// TwinCAT 3 PLC project DMAX
// Title: CalmarProdDmax
// Company: WIFAG-Polytype
// Author: Wifag//Polytype
// ProjectVersion: 2.0.2.24
// Description: All rights reserved (c) Wifag//Polytype, Fribourg/Switzerland (2021)
// ProgramVersion: 3.1.4023.0
// CompilerDefines: checks_in_libs
// libraries:
//   CalmarCommons, * (WIFAG-Polytype)
//   CalmarCompDevices, * (WIFAG-Polytype)
//   CalmarCompPrint, * (WIFAG-Polytype)
//   CalmarCompSystem, * (WIFAG-Polytype)
//   CalmarCompTcpIp, * (WIFAG-Polytype)
//   Tc2_EtherCAT, * (Beckhoff Automation GmbH)
//   Tc2_Math, * (Beckhoff Automation GmbH)
//   Tc2_Standard, * (Beckhoff Automation GmbH)
//   Tc2_System, * (Beckhoff Automation GmbH)
//   Tc2_TcpIp, * (Beckhoff Automation GmbH)
//   Tc2_Utilities, * (Beckhoff Automation GmbH)
//   Tc3_JsonXml, * (Beckhoff Automation GmbH)
//   VisuDialogs, * (System)
// project tree:
//   DUTs/Camera/ EN_CAMERA_TEACH.TcDUT, E_CameraDevice.TcDUT, E_CameraMode.TcDUT, E_DeformationType.TcDUT, ST_ADS_CAMERA.TcDUT, ST_CameraPoint.TcDUT, ST_CAMERA_CORRECTION_QV.TcDUT, ST_CAMERA_RESULT.TcDUT, ST_CAMERA_TEACH_QV.TcDUT, ST_CORRECTION_POINT.TcDUT, ST_TeachPoint.TcDUT
//   DUTs/ EN_MSG_LIST.TcDUT
//   / GlobalTextList.TcGTLO, Visualization Manager.TcVMO (not stored)
//   GVLs/ EC_DefGrid.TcGVL, GVL_Camera.TcGVL, GVL_Deformation.TcGVL
//   POUs/Machine/ExhaustSystem/ FB_ExhaustSystemPrint.TcPOU, _VISU_ExhaustSystemPrint.TcVIS
//   POUs/Machine/PowerControl/ FB_PowerControl.TcPOU, _VISU_PowerControl.TcVIS
//   POUs/Machine/UV_LED_Modul/ FB_UvLedModule.TcPOU, _VISU_UvLedModule.TcVIS
//   POUs/Print/Ads/ FB_ADS_CAMERA.TcPOU, FB_ADS_DVTSHEETALIGNMENT.TcPOU
//   POUs/Print/Camera/ FB_CameraBase.TcPOU, FB_CameraDummy.TcPOU, FB_CameraTcpIp.TcPOU, FB_CameraTrigger.TcPOU, FB_LineCamera.TcPOU, FB_LineCamera106.TcPOU, FB_LineCamera76.TcPOU, FB_MarkCamera.TcPOU, FB_SystronCamera.TcPOU, FB_TcpIpComm.TcPOU, F_DeformationPointAcc_ToString.TcPOU, F_CamPoint_ToString.TcPOU, ImagePool.TcIPO (not stored), I_Camera.TcIO, I_CameraSink.TcIO, I_CameraTrigger.TcIO, I_CameraTriggerDevice.TcIO, _VISU_CameraBase.TcVIS, _VISU_CameraBaseSetting.TcVIS, _VISU_CameraTcpIp.TcVIS, _VISU_CameraTcpIpSetting.TcVIS, _VISU_CameraTrigger.TcVIS, _VISU_DeformationPoint.TcVIS, _VISU_LineCamera.TcVIS, _VISU_MarkCamera.TcVIS (not stored), _VISU_SystronCamera.TcVIS
//   POUs/Print/DefGrid/ E_DeformationStep.TcTLEO, FB_ContainerDefGrid.TcPOU, FB_CTManagerDefGrid.TcPOU, FB_DeformationPointFIFO.TcPOU, FB_DropSpeedComp.TcPOU, FB_FineAlignement.TcPOU, FB_ImageDeformation.TcPOU, FB_DefGridParamMediator.TcPOU, FB_PointCorr.TcPOU, FB_PrintOverview.TcPOU, FB_PrintPositionDmax.TcPOU, FB_ProdManager_DMAX.TcPOU, FB_PythonDeformation.TcPOU, FB_PythonInterface.TcPOU, FB_StartPositionDummy.TcPOU, FB_WorkerDefGrid.TcPOU, FB_WorkerDefGrid_Camera.TcPOU, FB_WorkerDefGrid_Deformation.TcPOU, FB_WorkerDefGrid_Delete.TcPOU, FB_WorkerDefGrid_Print.TcPOU, FB_WorkerDefGrid_Python.TcPOU, FB_WorkerDefGrid_Verify.TcPOU, F_EncoderSpeedComp.TcPOU, F_MeterToSubPixelReal.TcPOU (not stored), I_DeformationHandler.TcIO, I_GridPointCorrection.TcIO, I_ParamMediator.TcIO, I_ProdManager.TcIO, ST_CameraGridSettings.TcDUT, ST_CameraPointTbl.TcDUT (not stored), ST_DeformationPointTbl.TcDUT, ST_WorkerDefGrid_CTData.TcDUT
//   POUs/Print/DefGrid/_Test/ E_GridTypeSelection.TcTLEO, Txt_GridTypeSelection.TcTLO
//   POUs/Print/DefGrid/_VISU_Templates/ E_DeformationType.TcTLO, _VISU_ContainerDefGrid.TcVIS, _VISU_CTsFlow.TcVIS, _VISU_DefGridTable.TcVIS, _VISU_FineAlignment.TcVIS, _VISU_GridPointView.TcVIS (not stored), _VISU_ImageDeformation.TcVIS (not stored), _VISU_PlacementXY.TcVIS (not stored), _VISU_PlacementXY_cross.TcVIS (not stored), _VISU_PrintPositionDmax.TcVIS (not stored), _VISU_DropSpeedComp_Setup.TcVIS, _VISU_StartPositionDummy.TcVIS (not stored), _VISU_WorkerDefGrid.TcVIS (not stored), _VISU_WorkerDefGrid_Camera.TcVIS (not stored), _VISU_WorkerDefGrid_Deformation.TcVIS (not stored), _VISU_WorkerDefGrid_Delete.TcVIS (not stored), _VISU_WorkerDefGrid_Print.TcVIS (not stored), _VISU_WorkerDefGrid_Python.TcVIS (not stored), _VISU_WorkerDefGrid_small.TcVIS (not stored), _VISU_WorkerDefGrid_Verify.TcVIS (not stored)
//   POUs/Print/ FB_SheetDetectSupervision.TcPOU, ST_SheetDetectSupervisionPar.TcDUT
//   Version/ Global_Version.TcGVL

// ---- DUTs/Camera/EN_CAMERA_TEACH.TcDUT
TYPE EN_CAMERA_TEACH :
(*************************************************************************************************)
(*  FILENAME:    EN_CAMERA_TEACH                                                                 *)
(*  PROJECT:     CALMAR PUPLC                                                                    *)
(*  COPYRIGHT:   All rights reserved (c) Wifag//Polytype, Fribourg/Switzerland (2018)            *)
(*  ENVIRONMENT: TwinCAT PLC                                                                     *)
(*  VERSION:     <version>                                                                       *)
(*************************************************************************************************)
(*  DESCRIPTION:                                                                   <description> *)
(*    Enumeration for camera teach.                                                              *)
(*                                                                                </description> *)
(*************************************************************************************************)

(
  eTeachInit         := 0,
  eTeachStart        := 1,
  eTeachCompleted    := 2,
  eTeachCanceled     := 3,
  eTeachError        := 4
);
END_TYPE

// ---- DUTs/Camera/E_CameraDevice.TcDUT
{attribute 'qualified_only'}
{attribute 'strict'}
{attribute 'to_string'}
TYPE E_CameraDevice :
(
  SheetDetect              := 0,   // SheetDetect
  PrintMark                := 1,   // PrintMark
  Scanner                  := 2,   // Scanner
  ScannerWithoutBackground := 3    // ScannerWithoutBackground
);
END_TYPE

// ---- DUTs/Camera/E_CameraMode.TcDUT
{attribute 'qualified_only'}
{attribute 'strict'}
{attribute 'to_string'}
TYPE E_CameraMode :
(
  NoCorrection := 0,   // NoCorrection
  XYR          := 1,   // XYR
  Live         := 2,   // Live deformation
  Trend        := 3,   // Live deformation with trend
  Auto         := 4    // Auto
);
END_TYPE

// ---- DUTs/Camera/E_DeformationType.TcDUT
{attribute 'qualified_only'}
{attribute 'to_string'}
TYPE E_DeformationType :
(
  NoDeformation   := 0,   // NoCorrection
  ScriptGrid      := 1,   // Py script (live)
  ScriptGridTrend := 2,   // Py script (live with trend)
  LocalMarks1D    := 3    // Plc generated with 1D marks
)  UINT;
END_TYPE

// ---- DUTs/Camera/ST_ADS_CAMERA.TcDUT
TYPE ST_ADS_CAMERA :
(*************************************************************************************************)
(*  FILENAME:    ST_ADS_CAMERA                                                                   *)
(*  PROJECT:     CALMAR PUPLC                                                                    *)
(*  COPYRIGHT:   All rights reserved (c) Wifag//Polytype, Fribourg/Switzerland (2018)            *)
(*  ENVIRONMENT: TwinCAT PLC                                                                     *)
(*  VERSION:     <version>                                                                       *)
(*************************************************************************************************)
(*  DESCRIPTION:                                                                   <description> *)
(*    ADS structure for camera (Systron, QualiVision).                                           *)
(*                                                                                </description> *)
(*************************************************************************************************)

STRUCT
  iO_Version                : UINT    := 010300;  (*1.3.0*)
  aO_Type                   : STRING := 'Camera';
  aO_Name                   : STRING := 'Camera';
  sO_Message                : ST_ADS_MSG_IF;

  (*In*)
  bI_Enable                 : BOOL := TRUE;      (*Enable this device*)

  eI_CameraDevice           : E_CameraDevice;    (*Camera device*)
  eI_CameraMode             : E_CameraMode;      (*Camera mode*)

  eI_TeachProgress          : EN_CAMERA_TEACH;   (*Teach progress*)
  sI_TeachPointsQV          : ARRAY[1..GVL_Camera.cC_QUALIVISION_MAX_NB_MARKS] OF ST_CAMERA_TEACH_QV;
  
  sI_CorrectionPointIndication: ARRAY[1..4] OF ST_CORRECTION_POINT;

  (*Out*)
  iO_MaxNbMarksQV           : INT := GVL_Camera.cC_QUALIVISION_MAX_NB_MARKS; 
  sO_PointsReadQV           : ST_COMMAND_PLC;    (*New points read by QualiVision*)
  iO_AvailableNbReadPointQV : INT; 
  sO_ReadPointsQV           : ARRAY[1..GVL_Camera.cC_QUALIVISION_MAX_NB_MARKS] OF ST_CAMERA_CORRECTION_QV;

END_STRUCT
END_TYPE

// ---- DUTs/Camera/ST_CameraPoint.TcDUT
TYPE ST_CameraPoint :
STRUCT
  (*Valus from camera [px/4800dpi]*)
  id                  : UDINT := 0;     (*mark id*)
  x_ref               : DINT := 0;      (*Referenz x deviation [px/4800dpi]*)
  y_ref               : DINT := 0;      (*Referenz y deviation [px/4800dpi]*)
  lx                  : DINT := 0;      (*Referenz in picture x deviation [px/4800dpi]*)
  ly                  : DINT := 0;      (*Referenz in picture y deviation [px/4800dpi]*)
  valid               : BOOL := FALSE;  (*TRUE = PASS, FALSE = FAIL*)
  x                   : DINT := 0;      (*x deviation [px/4800dpi]*)
  y                   : DINT := 0;      (*y deviation [px/4800dpi]*)
END_STRUCT
END_TYPE

// ---- DUTs/Camera/ST_CAMERA_CORRECTION_QV.TcDUT
TYPE ST_CAMERA_CORRECTION_QV :
(*************************************************************************************************)
(*  FILENAME:    ST_CAMERA_CORRECTION_QV                                                         *)
(*  PROJECT:     CALMAR PUPLC                                                                    *)
(*  COPYRIGHT:   All rights reserved (c) Wifag//Polytype, Fribourg/Switzerland (2016)            *)
(*  ENVIRONMENT: TwinCAT PLC                                                                     *)
(*  VERSION:     <version>                                                                       *)
(*************************************************************************************************)
(*  DESCRIPTION:                                                                   <description> *)
(*    Correction of smart camera QualiVision for PUC.                                            *)
(*                                                                                </description> *)
(*************************************************************************************************)

STRUCT
  (*PUC correction points [mm]*)
  valid               : BOOL := FALSE;  (*TRUE = PASS, FALSE = FAIL*)
  PaddingByte01       : BYTE;           (*PUC needs it for stream reading. TC3 uses 8 byte alignment.*)
  PaddingByte02       : BYTE;           (*PUC needs it for stream reading. TC3 uses 8 byte alignment.*)
  PaddingByte03       : BYTE;           (*PUC needs it for stream reading. TC3 uses 8 byte alignment.*)
  x_origin            : REAL := 0;      (*Referenz x origin [mm]*)
  y_origin            : REAL := 0;      (*Referenz y origin [mm]*)
  x_correction        : REAL := 0;      (*x correction [mm]*)
  y_correction        : REAL := 0;      (*y correction [mm]*)
  PaddingBytes04      : REAL;           (*PUC needs it for stream reading. TC3 uses 8 byte alignment.*)
END_STRUCT
END_TYPE

// ---- DUTs/Camera/ST_CAMERA_RESULT.TcDUT
TYPE ST_CAMERA_RESULT :
(*************************************************************************************************)
(*  FILENAME:    ST_CAMERA_RESULT.EXP                                                            *)
(*  PROJECT:     CALMAR PUPLC                                                                    *)
(*  COPYRIGHT:   All rights reserved (c) Wifag//Polytype, Fribourg/Switzerland (2016)            *)
(*  ENVIRONMENT: TwinCAT PLC                                                                     *)
(*  VERSION:     <version>                                                                       *)
(*************************************************************************************************)
(*  DESCRIPTION:                                                                   <description> *)
(*    Output of smart camera Systron.                                                            *)
(*                                                                                </description> *)
(*************************************************************************************************)

STRUCT
  x_ref               : REAL := 0;      (*Referenz x deviation [mm]*)
  y_ref               : REAL := 0;      (*Referenz y deviation [mm]*)
  valid               : BOOL := TRUE;   (*TRUE = PASS, FALSE = FAIL*)
  x                   : REAL := 0;      (*x deviation [mm]*)
  y                   : REAL := 0;      (*y deviation [mm]*)
END_STRUCT
END_TYPE

// ---- DUTs/Camera/ST_CAMERA_TEACH_QV.TcDUT
TYPE ST_CAMERA_TEACH_QV :
(*************************************************************************************************)
(*  FILENAME:    ST_CAMERA_TEACH_QV                                                              *)
(*  PROJECT:     CALMAR PUPLC                                                                    *)
(*  COPYRIGHT:   All rights reserved (c) Wifag//Polytype, Fribourg/Switzerland (2016)            *)
(*  ENVIRONMENT: TwinCAT PLC                                                                     *)
(*  VERSION:     <version>                                                                       *)
(*************************************************************************************************)
(*  DESCRIPTION:                                                                   <description> *)
(*    Teach points for smart camera QualiVision from PUC.                                        *)
(*                                                                                </description> *)
(*************************************************************************************************)

STRUCT
  x_ref_Print         : REAL := 0;      (*Referenz x deviation [mm]*)
  y_ref_Print         : REAL := 0;      (*Referenz y deviation [mm]*)
END_STRUCT
END_TYPE

// ---- DUTs/Camera/ST_CORRECTION_POINT.TcDUT
TYPE ST_CORRECTION_POINT :
(*************************************************************************************************)
(*  FILENAME:    ST_CORRECTION_POINT                                                             *)
(*  PROJECT:     CALMAR PUPLC                                                                    *)
(*  COPYRIGHT:   All rights reserved (c) Wifag//Polytype, Fribourg/Switzerland (2021)            *)
(*  ENVIRONMENT: TwinCAT PLC                                                                     *)
(*  VERSION:     <version>                                                                       *)
(*************************************************************************************************)
(*  DESCRIPTION:                                                                   <description> *)
(*    PUC correction point indication provided from job, written at print start.                 *)
(*                                                                                </description> *)
(*************************************************************************************************)

STRUCT
  x        : REAL := 0;      (*Correction indication x [mm]*)
  y        : REAL := 0;      (*Correction indication y [mm]*)
  posx     : REAL := 0;      (*Correction location in x [mm]*)
  posy     : REAL := 0;      (*Correction location in y [mm]*)
END_STRUCT
END_TYPE

// ---- DUTs/Camera/ST_TeachPoint.TcDUT
TYPE ST_TeachPoint :
STRUCT
  (*Valus for printer [mm]*)
  id                  : UDINT;           (*point id*)
  x_ref_Print         : LREAL := 0;      (*Referenz x deviation [mm]*)
  y_ref_Print         : LREAL := 0;      (*Referenz y deviation [mm]*)
  x_teach_Print       : LREAL := 0;      (*Teach x deviation [mm]*)
  y_teach_Print       : LREAL := 0;      (*Teach y deviation [mm]*)
  x_Print             : LREAL := 0;      (*x deviation [mm]*)
  y_Print             : LREAL := 0;      (*y deviation [mm]*)
  valid               : BOOL  := FALSE;  (**)
END_STRUCT
END_TYPE

// ---- DUTs/EN_MSG_LIST.TcDUT
TYPE EN_MSG_LIST :
(*************************************************************************************************)
(*  FILENAME:    EN_MSG_LIST.EXP                                                                 *)
(*  PROJECT:     CALMAR PUPLC                                                                    *)
(*  COPYRIGHT:   All rights reserved (c) Wifag//Polytype, Fribourg/Switzerland (2016)            *)
(*  ENVIRONMENT: TwinCAT PLC                                                                     *)
(*  VERSION:     <version>                                                                       *)
(*************************************************************************************************)
(*  DESCRIPTION:                                                                   <description> *)
(*     This block containts the global list for all messages used by `FB_MESSAGE`.               *)
(*                                                                                </description> *)
(*************************************************************************************************)
(
  // start at                       eCStag_MSG_BASE := 10000,
  eC_STAG_CAM_NOTAVAIL                              :=10000,  (*CameraNotAvailable*)
  eC_STAG_CAM_MODE_NOTSUPPORTED                     :=10001,  (*CameraModeNotSupported*)
  eC_STAG_CAM_NOTENGOUGH_TEACH_POINTS               :=10002,  (*CameraNotEnoughTeachPoints*)
  eC_STAG_DEF_SCRIPT_NOT_RUNNING                    :=10003,  (*DeformationScriptNotRunning*)
  eC_STAG_CAM_TEACH_ERROR                           :=10004,  (*CameraTeachError*)
  eC_STAG_IMAGELENGTH_NOT_SUPPORTED                 :=10005,  (*ImageLengthNotSupported*)
  eC_STAG_DEFORMATION_LIMITED                       :=10006   (*DeformationWasLimited (Warning)*)
);
END_TYPE

// ---- POUs/Print/DefGrid/E_DeformationStep.TcTLEO
{attribute 'qualified_only'}
{attribute 'strict'}
{attribute 'to_string'}
TYPE E_DeformationStep :
(
  nothing := 0,
  createdScriptContainer := 1,
  cameraStarted := 2,
  cameraDone := 3,
  gridStarted := 4
);
END_TYPE

// ---- POUs/Print/DefGrid/ST_CameraGridSettings.TcDUT
TYPE ST_CameraGridSettings :
STRUCT
  bValid            : BOOL;   // ?
  eCameraMode       : E_CameraMode;
  eDeformationType  : E_DeformationType;  // selected deformation type based on selecte camera and settings
  fGridFeaturePitch : LREAL;  // feature grid picth (cam frame width) [px]
  fDetectToCam      : LREAL;  // distance between detection and camera [m]
END_STRUCT
END_TYPE

// ---- POUs/Print/DefGrid/ST_DeformationPointTbl.TcDUT
(*
  Table representation of a point
*)
TYPE ST_DeformationPointTbl :
STRUCT
  bSet          : BOOL;
  tTime         : T_DCTIME64;
  sPoint        : ST_DeformationPointAccurate;
END_STRUCT
END_TYPE

// ---- POUs/Print/DefGrid/ST_WorkerDefGrid_CTData.TcDUT
// workers additional data for all attached CTs
TYPE ST_WorkerDefGrid_CTData :
STRUCT
  fPosRelToAttach : LREAL;    // ct relative position to attach
  nChargedCols : UDINT;       // number of streamed columns of this ct
  nXS : DINT;                 // XS print start position
END_STRUCT
END_TYPE

// ---- POUs/Print/DefGrid/_Test/E_GridTypeSelection.TcTLEO
{attribute 'qualified_only'}
{attribute 'strict'}
{attribute 'to_string'}
TYPE E_GridTypeSelection :
(
  Default             := 0,  // Default deformation based on cam points
  None                := 1,  // No deformation calculated all dx/dy=0
  Test_AllDxFactor    := 2,  // Dx constant for all = factor
  Test_AllDyFactor    := 3,  // Dy constant for all = factor
  Test_DyColFactor    := 4,  // Dy = col * factor (changes by column)
  Test_DxColFactor    := 5,  // Dx = col * factor (changes by column)
  Test_Dx_Row1OnlyFactor := 6   // dx factor only on row1 (test BOF)
) UINT := Default ;
END_TYPE

// ---- POUs/Print/ST_SheetDetectSupervisionPar.TcDUT
TYPE ST_SheetDetectSupervisionPar :
STRUCT
  bR_Enable                   : BOOL  := TRUE;
  fR_SheetDetectDistance01    : LREAL := 0.656;  //[m]
  fR_SheetDetectRange01_m     : REAL  := 0.03;   //[m]
  nR_SheetDetectRange01_SubPx : DINT;            //[SubPx]
  fR_SheetDetectDistance02    : LREAL := 1.031;  //[m]
  fR_SheetDetectRange02_m     : REAL  := 0.03;   //[m]
  nR_SheetDetectRange02_SubPx : DINT;            //[SubPx]
END_STRUCT
END_TYPE

// ---- GVLs/EC_DefGrid.TcGVL
{attribute 'qualified_only'}
(*
  Calmar Error Codes - CalmarProductsSteinemann library
*)
VAR_GLOBAL
  // base
  _ecBase        : UDINT := CalmarCommons.ErrorCodes.lCalmar_base;
  _ecProjBase    : UDINT := _ecBase OR 16#00150000;

  // DefGrid error
  ecDefGrid_DefGridError : T_ErrDef(Id:=_ecProjBase OR 16#001, Code:='GridError', Desc:='Error in script happened');
  ecDefGrid_DefGridAbort : T_ErrDef(Id:=_ecProjBase OR 16#002, Code:='GridAbort', Desc:='Deformation aborted');
  
  // Camera errors
  ecDefGrid_CamNotAvailable : T_ErrDef(Id:=_ecProjBase OR 16#010, Code:='CamNotAvailable', Desc:='Desired camera not available');
  
  // end (verify to not overflow the group range!)
END_VAR

// ---- GVLs/GVL_Camera.TcGVL
{attribute 'qualified_only'}
VAR_GLOBAL CONSTANT
  cMaxNbMarks                   : UDINT := 200;     (*Max number of QualiVision marks*)
  cMaxNbSectors                 : UDINT := 50;      (*Max number of QualiVision sectors*)
  cC_QUALIVISION_MAX_NB_MARKS   : BYTE  := 10;      (*Max number of QualiVision marks*)
  nC_NbCamErrors                : UDINT := 10;
END_VAR

// ---- GVLs/GVL_Deformation.TcGVL
{attribute 'qualified_only'}
VAR_GLOBAL
// moved to CompPrint FB_PH
  //  nC_GridPitch_X  : UDINT := 1024;    // GRID: distance between grid point in y [px] (FPGA definition)
  //  nC_GridPitch_Y  : UDINT := 2048;    // GRID: distance between grid point in y [px] (FPGA definition)
  //  nC_GridRoiRows  : UINT  := 3;       // ROI: [1024=4,  2048=3] number of roi rows per head (FPGA definition) 
  //  nC_GridRoiCols  : UINT  := 85;      // ROI: [1024=62, 2048=85] number of roi columns per head (FPGA definition) 

  nC_DefaultGridPitch_X  : UDINT := 1024;    // GRID: (default if unknown in hw) distance between grid point in y [px] (FPGA definition)
  nC_DefaultGridPitch_Y  : UDINT := 2048;    // GRID: (default if unknown in hw) distance between grid point in y [px] (FPGA definition)
  nC_GridSubReso  : UDINT := 10;      // sub resolution of grid definitions (script handling)
  bC_UsePUDeformation : BOOL := TRUE;   // enable calculation of PU deformation/correction
END_VAR

// ---- Version/Global_Version.TcGVL
{attribute 'TcGenerated'}
{attribute 'no-analysis'}
{attribute 'linkalways'}
// This function has been automatically generated from the project information.
VAR_GLOBAL CONSTANT
	{attribute 'const_non_replaced'}
	stLibVersion_CalmarProductSteinemann : ST_LibVersion := (iMajor := 3, iMinor := 0, iBuild := 4, iRevision := 0, nFlags := 0, sVersion := '3.0.4');
END_VAR

// ---- POUs/Print/Camera/I_Camera.TcIO
INTERFACE I_Camera

METHOD ActivateCam : BOOL
VAR_INPUT
  iCameraSink : I_CameraSink;
END_VAR
END_METHOD

(*
  Activate/Deactivate camera trigger device
*)
PROPERTY bEnableTrigger : BOOL
SET
END_SET
END_PROPERTY

(*
  Activate/Deactivate camera manual teach mode
*)
PROPERTY bManualTeach : BOOL
SET
END_SET
END_PROPERTY

{attribute 'monitoring':='call'}
PROPERTY bSimulate : BOOL
GET
END_GET
SET
END_SET
END_PROPERTY

METHOD DeactivateCam : BOOL
VAR_INPUT
  iSink : I_CameraSink;
END_VAR
END_METHOD

{attribute 'monitoring':='call'}
PROPERTY ABSTRACT eCameraMode : E_CameraMode
GET
END_GET
END_PROPERTY

{attribute 'monitoring':='call'}
PROPERTY ABSTRACT eDeviceType : E_CameraDevice
GET
END_GET
END_PROPERTY

{attribute 'monitoring':='call'}
PROPERTY fCameraToPrintOffset : LREAL
GET
END_GET
END_PROPERTY

{attribute 'monitoring':='call'}
PROPERTY fDetectToCameraOffset : LREAL
GET
END_GET
END_PROPERTY

{attribute 'monitoring':='call'}
// camera frame size in [px]
PROPERTY fFrameLength : LREAL
GET
END_GET
SET
END_SET
END_PROPERTY

{attribute 'monitoring':='call'}
(*Image Length/Depth in [m]*)
PROPERTY fImageLength : LREAL
GET
END_GET
SET
END_SET
END_PROPERTY

{attribute 'monitoring':='call'}
(*Image Width in [m]*)
PROPERTY fImageWidth : LREAL
GET
END_GET
SET
END_SET
END_PROPERTY

{attribute 'monitoring':='call'}
(*Substrate Length/Depth in [m]*)
PROPERTY fSubstrateLength : LREAL
GET
END_GET
SET
END_SET
END_PROPERTY

{attribute 'monitoring':='call'}
(*Substrate Width in [m]*)
PROPERTY fSubstrateWidth : LREAL
GET
END_GET
SET
END_SET
END_PROPERTY

{attribute 'monitoring':='call'}
PROPERTY fTriggerDistance : LREAL
GET
END_GET
SET
END_SET
END_PROPERTY

(*
  Get camera status.
  :return: TRUE if camera is ok
*)
METHOD GetCamStatus : BOOL  // Camera Ok?
VAR_OUTPUT
  bConnectionOK  : BOOL;    // Camera connected
  bTeachOk       : BOOL;    // Teach successful
  nTeachedPoints : UDINT;   // Teached points for this job
  nScannedPoints : UDINT;   // Scanned points on current CT
  bCamStarted    : BOOL;    // Camera trigger is active, cam started
  bCamDone       : BOOL;    // Camera finished on last CT
  bErrors        : ARRAY[1..GVL_Camera.nC_NbCamErrors] OF BOOL;  // generic error flag list
END_VAR
END_METHOD

METHOD mJobStart : BOOL
VAR_INPUT
END_VAR
END_METHOD

(*
  Set mode to camera.
  :return: TRUE if success
*)
METHOD setCameraMode : BOOL
VAR_INPUT
  eCameraMode : E_CameraMode;
END_VAR
END_METHOD

METHOD setMsgInterface : BOOL
VAR_INPUT
  pMsgConfig  : POINTER TO ST_MSG_CONFIG;
END_VAR
END_METHOD

{attribute 'monitoring':='call'}
PROPERTY sName : STRING
GET
END_GET
END_PROPERTY

{attribute 'monitoring':='call'}
PROPERTY sVisuName : STRING
GET
END_GET
END_PROPERTY

END_INTERFACE

// ---- POUs/Print/Camera/I_CameraSink.TcIO
{attribute 'monitoring':='call'}
INTERFACE I_CameraSink

METHOD AddCamPoint : BOOL
VAR_INPUT
	sDeformationPoint	: ST_DeformationPointAccurate;
END_VAR
END_METHOD

METHOD AddTeachPoint : BOOL
VAR_INPUT
  sTeachPoint : ST_DeformationPointAccurate;
END_VAR
END_METHOD

(*
  Event cam done "detecting points", sheet/repeate done.
  Called after last point will be streamed to same CT.
*)
METHOD CamDone : BOOL
END_METHOD

(*
  Event cam started "detecting points".
  Is called before streaming cam points.
*)
METHOD CamStarted
VAR_INPUT
  nX0 : DINT; // detected start position
END_VAR
END_METHOD

// Detected "real" image lenght [m]
PROPERTY fPrintLengthEffective : LREAL
SET
END_SET
END_PROPERTY

END_INTERFACE

// ---- POUs/Print/Camera/I_CameraTrigger.TcIO
INTERFACE I_CameraTrigger

PROPERTY bManualTeach : BOOL
GET
END_GET
SET
END_SET
END_PROPERTY

METHOD Disable : BOOL
VAR_INPUT
END_VAR
END_METHOD

METHOD Enable : BOOL
VAR_INPUT
  iCam : I_CameraTriggerDevice;
  bUseCameraTrigger : BOOL; //Generate camera trigger
  bUseCameraTriggerFeedback : BOOL; //Use feedback as trigger?
END_VAR
END_METHOD

METHOD SetSubstrateLength
VAR_INPUT
  fSubstrateLength : LREAL;
END_VAR
END_METHOD

END_INTERFACE

// ---- POUs/Print/Camera/I_CameraTriggerDevice.TcIO
INTERFACE I_CameraTriggerDevice

METHOD CamTrigger
VAR_INPUT
  bOk             : BOOL;     // trigger is ok
	nPos            : DINT;     // camera triggered position
  nPosDeviation   : DINT;     // camera started deviation
  nX0             : DINT;     // detected position sheet/repetition
END_VAR
END_METHOD

METHOD CamTriggerDone
VAR_INPUT
END_VAR
END_METHOD

{attribute 'monitoring':='call'}
PROPERTY fTriggerDistance : LREAL
GET
END_GET
END_PROPERTY

PROPERTY fTriggerPulseLength : LREAL
GET
END_GET
END_PROPERTY

END_INTERFACE

// ---- POUs/Print/DefGrid/I_DeformationHandler.TcIO
INTERFACE I_DeformationHandler

METHOD DeleteCachedCt : BOOL
VAR_INPUT
  iCT              : I_CT;
END_VAR
END_METHOD

END_INTERFACE

// ---- POUs/Print/DefGrid/I_GridPointCorrection.TcIO
INTERFACE I_GridPointCorrection

(*
  Apply correction to gridPoint
*)
METHOD updateCorrection : BOOL
VAR_INPUT
  pPoint : POINTER TO ST_DeformationPointAccurate;
END_VAR
END_METHOD

END_INTERFACE

// ---- POUs/Print/DefGrid/I_ParamMediator.TcIO
INTERFACE I_ParamMediator

PROPERTY sCameraGridSettings : ST_CameraGridSettings
GET
END_GET
END_PROPERTY

PROPERTY sDeformationGridSettings : ST_DefGridSettings
GET
END_GET
END_PROPERTY

END_INTERFACE

// ---- POUs/Print/DefGrid/I_ProdManager.TcIO
INTERFACE I_ProdManager

END_INTERFACE

// ---- POUs/Machine/ExhaustSystem/FB_ExhaustSystemPrint.TcPOU
FUNCTION_BLOCK FB_ExhaustSystemPrint
VAR_INPUT
  bI_FUReady                         AT %I* : BOOL;   (*FU ready*)
  iI_VacuumMeasurement               AT %I* : UINT;   (*Analog input: vacuum measurement*)
  bPrintActive                              : BOOL;   (*Printing active*)
END_VAR

VAR_OUTPUT
  bO_FUActivate                      AT %Q* : BOOL;   (*FU activation*)
  OnExhaustSetpoint                  AT %Q* : UINT;   (*Analog output: pump setpoint*)

  bExhaustError                             : BOOL;   (*Exhaust system ok and ready*)
  // detailed status (for messages)
  bFUReady                                  : BOOL;   (*FU ready*)
  bVacuumWarningLevel                       : BOOL;   (*Vacuum warning level reached*)
  bVacuumErrorLevel                         : BOOL;   (*Vacuum error level reached*)
END_VAR

VAR
  iL_Counter                                : INT;    (*Basic counter*)
  bMappingChecked                           : BOOL;   (*Checked mapped variable status*)
  bMapping_FUReady_Done                     : BOOL;   (*FUReady is mapped*)
  
  fb_TofFUOffDelay                          : TOF;    (*FU off delay*)
  fb_TonVacuumCheckDelay                    : TON;    (*Vacuum check delay*)

  fL_VacuumAnalogLevelMBar                  : REAL;   (*Actual value analog-input in mBar*)
END_VAR

VAR PERSISTENT
  tR_FUOffDelay                             : TIME := T#3M;   (*FU off delay time*)
  tR_VacuumCheckDelay                       : TIME := T#10S;  (*Vacuum check delay time*)

  iR_VacuumAnalogMinDigit                   : UINT := 0;      (*Min value analog-input in digit*)
  iR_VacuumAnalogMaxDigit                   : UINT := 32767;  (*Max value analog-input in digit*)
  fR_VacuumAnalogMinMBar                    : REAL := 0;      (*Min value analog-input in mBar*)
  fR_VacuumAnalogMaxMBar                    : REAL := 50.0;   (*Max value analog-input in mBar*)
  fR_VacuumWarningLevelMBar                 : REAL := 20.0;   (*Warning level in mBar*)
  fR_VacuumErrorLevelMBar                   : REAL := 10.0;   (*Error level in mBar*)

  iR_VacuumPumpSetPercent                   : UINT := 0;      (*Pump setpoinr [%]*)
  iR_VacuumPumpSetpointMaxDigit             : UINT := 13762;  (*Max value analog-output in digit, max pump = 4.2V*)
END_VAR

// mapping check
IF NOT bMappingChecked THEN checkMapping(); END_IF
IF NOT bMapping_FUReady_Done THEN bI_FUReady := TRUE; END_IF    // if not mapped is ready


bFUReady := bI_FUReady;  // AND bO_FUActivate?

fb_TofFUOffDelay(IN := bPrintActive, PT := tR_FUOffDelay);    // turn-off delay
bO_FUActivate := fb_TofFUOffDelay.Q;

fL_VacuumAnalogLevelMBar := UINT_TO_REAL(iI_VacuumMeasurement) * fR_VacuumAnalogMaxMBar / iR_VacuumAnalogMaxDigit;

fb_TonVacuumCheckDelay(IN := bO_FUActivate, PT := tR_VacuumCheckDelay);   // delay for vacum measurement
IF fb_TonVacuumCheckDelay.Q THEN
  // check levels and set waring/error
  bVacuumWarningLevel := fL_VacuumAnalogLevelMBar < fR_VacuumWarningLevelMBar;
  bVacuumErrorLevel   := fL_VacuumAnalogLevelMBar < fR_VacuumErrorLevelMBar;
END_IF


bExhaustError := NOT bFUReady OR (bVacuumErrorLevel AND bO_FUActivate);

OnExhaustSetpoint := REAL_TO_UINT(UINT_TO_REAL(iR_VacuumPumpSetpointMaxDigit) / 100 * iR_VacuumPumpSetPercent);

METHOD PRIVATE checkMapping
VAR_INPUT
END_VAR
bMapping_FUReady_Done := F_GetMappingStatus(p:=ADR(bI_FUReady), n:=SIZEOF(bI_FUReady)) > EPlcMappingStatus.MS_Unmapped;

bMappingChecked := TRUE;
END_METHOD

METHOD mAckError : BOOL
VAR_INPUT
END_VAR
bVacuumWarningLevel := FALSE;
bVacuumErrorLevel   := FALSE;
END_METHOD

END_FUNCTION_BLOCK

// ---- POUs/Machine/PowerControl/FB_PowerControl.TcPOU
(*
  PowerSupply control (WAGO Epsitron)
  NOTE: has direct mapped I/Os
*)
FUNCTION_BLOCK FB_PowerControl EXTENDS T_NamedBase
VAR_OUTPUT
  bO_AllFuseOk        : BOOL;
  bO_AllEpsitronOk    : BOOL;
  bO_AllInputOk       : BOOL;
END_VAR
VAR
  i : UDINT;
  
  // Commands
  bAckMsg : BOOL;
  
  // Epsitron Controls
  fbEpsitronFuseControl                     : ARRAY[1..nMaxEpsitrons] OF FB_EpsitronFuseControl;   // internal instances of epsitrons
  // list of epsitron for view & global control
  pEpsitronsInst                            : ARRAY[1..nMaxEpsitrons] OF POINTER TO FB_EpsitronFuseControl;   // list
  bEpsitronsAllChOk                         : ARRAY[1..nMaxEpsitrons] OF BOOL;
  nEpsitronsRegistered                      : UDINT := 0;
  nEpsitronViewSel                          : UDINT := 1;
  
  // Fuse (I/O) supervision
  nFuseInputsRegistered                     : UDINT;
  aFuseNames                                : ARRAY[1..nMaxFuseInputs] OF STRING;
  pFuseInputs                               : ARRAY[1..nMaxFuseInputs] OF POINTER TO BOOL;
  nFuseViewSel                              : UDINT := 1;
END_VAR
VAR CONSTANT
  nMaxEpsitrons : UDINT := 10;
  nMaxFuseInputs : UDINT := 20;
END_VAR

bO_AllEpsitronOk := TRUE;
FOR i:=1 TO nEpsitronsRegistered DO
  IF pEpsitronsInst[i] <> 0 THEN
    pEpsitronsInst[i]^();
    
    bEpsitronsAllChOk[i] := NOT (   (pEpsitronsInst[i]^.iO_Channel1Status = 3)
                              OR (pEpsitronsInst[i]^.iO_Channel2Status = 3)
                              OR (pEpsitronsInst[i]^.iO_Channel3Status = 3)
                              OR (pEpsitronsInst[i]^.iO_Channel4Status = 3));

    
    bO_AllEpsitronOk := bO_AllEpsitronOk AND bEpsitronsAllChOk[i];
  END_IF
END_FOR

// I/O inputs
bO_AllInputOk := TRUE;
FOR i:=1 TO nFuseInputsRegistered DO
  IF pFuseInputs[i] <> 0 THEN
    bO_AllInputOk := bO_AllInputOk AND pFuseInputs[i]^;
  END_IF
END_FOR       

// output
bO_AllFuseOk := bO_AllEpsitronOk AND bO_AllInputOk;
 
// Acknowledge error
IF bAckMsg THEN  bAckMsg := FALSE;
  FOR i:=1 TO nEpsitronsRegistered DO
    pEpsitronsInst[i]^.mAckError();
	END_FOR
END_IF

METHOD ackError
bAckMsg := TRUE;
END_METHOD

(*
  Register configuration for an epsitron directly I/O mapped into this FB.
*)
METHOD registerEpsitron : BOOL
VAR_INPUT
  nInstIdx : UDINT;     // array instance index
  aName    : STRING;    // Epsitron name
  aNameCh1 : STRING;    // name of channel1
  aNameCh2 : STRING;    // name of channel2
  aNameCh3 : STRING;    // name of channel3
  aNameCh4 : STRING;    // name of channel4
END_VAR
IF nInstIdx > nMaxEpsitrons OR nInstIdx = 0      THEN LogError(F_Concat2('registerEpsitron: Invalid index, ignore: ', aName)); END_IF
IF fbEpsitronFuseControl[nInstIdx].aI_Name <> '' THEN LogError(F_Concat2('registerEpsitron: Already configured, ignore: ', aName)); END_IF
IF nEpsitronsRegistered >= nMaxEpsitrons         THEN LogError(F_Concat2('registerEpsitron: Too many already registered, ignore: ', aName)); END_IF
IF aName = ''                                  THEN LogWarning(F_Concat2('registerEpsitron: No name given', '')); END_IF

fbEpsitronFuseControl[nInstIdx].aI_Name := aName;
fbEpsitronFuseControl[nInstIdx].aI_NameChannel1 := aNameCh1;
fbEpsitronFuseControl[nInstIdx].aI_NameChannel2 := aNameCh2;
fbEpsitronFuseControl[nInstIdx].aI_NameChannel3 := aNameCh3;
fbEpsitronFuseControl[nInstIdx].aI_NameChannel4 := aNameCh4;

nEpsitronsRegistered := nEpsitronsRegistered + 1;
pEpsitronsInst[nEpsitronsRegistered] := ADR(fbEpsitronFuseControl[nInstIdx]);

registerEpsitron := TRUE;
END_METHOD

METHOD registerIO : BOOL
VAR_INPUT
  aName  : STRING;              // name of fuse (bool) input
  pInput : POINTER TO BOOL;     // I/O value pointer
END_VAR
IF nFuseInputsRegistered >= nMaxFuseInputs  THEN LogError(F_Concat2('registerIO: Too many already registered, ignore: ', aName)); END_IF
IF pInput = 0                               THEN LogError(F_Concat2('registerIO: Invalid pointer given, ignore: ', aName)); END_IF
IF aName = ''                               THEN LogWarning(F_Concat2('registerIO: No name given', '')); END_IF

nFuseInputsRegistered := nFuseInputsRegistered + 1;
aFuseNames[nFuseInputsRegistered]  := aName;
pFuseInputs[nFuseInputsRegistered] := pInput;

registerIO := TRUE;
END_METHOD

END_FUNCTION_BLOCK

// ---- POUs/Machine/UV_LED_Modul/FB_UvLedModule.TcPOU
FUNCTION_BLOCK FB_UvLedModule IMPLEMENTS I_DeviceBase
VAR_INPUT
  IbReady                  AT%I* : BOOL;
END_VAR

VAR_OUTPUT
  ObEnableHigh             AT%Q* : BOOL;
  ObLowIntenseMode         AT%Q* : BOOL;
  ObDisableLeft            AT%Q* : BOOL;
  ObDisableRight           AT%Q* : BOOL;
  OnIntensitySetpoint      AT%Q* : WORD;  (*Setpoint for intensity control  [digit]*)
END_VAR

VAR
  _bActivate                     : BOOL;
  _sName                         : STRING := '';
  _nColorRGB                     : UDINT;
  _sColorName                    : STRING := 'undef';    (*color name*)
END_VAR

VAR CONSTANT
  CnAnalogMinDigit               : DINT := 0;      (*Min value analog-output in digit*)
  CnAnalogMaxDigit               : DINT := 32767;  (*Max value analog-output in digit*)
  CnMinIntensitySetpoint         : DINT := 5;      (*Min setpoint for intensity control [%]*)
  CnMaxIntensitySetpoint         : DINT := 100;    (*Max setpoint for intensity control [%]*)
END_VAR

VAR PERSISTENT
  RbLowIntenseMode               : BOOL := FALSE;  (*Visu: set low intense mode*)
  RbDisableLeft                  : BOOL := FALSE;  (*Visu: disable left SLM*)
  RbDisableRight                 : BOOL := FALSE;  (*Visu: disable right SLM*)
  RnIntensitySetpoint            : DINT := 20;     (*Visu: setpoint for intensity control [%]*)
END_VAR

(*Set outputs*)
ObEnableHigh        := _bActivate;
ObLowIntenseMode    := RbLowIntenseMode;
ObDisableLeft       := RbDisableLeft;
ObDisableRight      := RbDisableRight;
OnIntensitySetpoint := DINT_TO_WORD(CnAnalogMaxDigit * RnIntensitySetpoint / 100);  (*Setpoint [digit]*)

METHOD Init : BOOL
VAR_INPUT
  nColorRGB    : UDINT;     (*color RGB*)
  sColorName   : STRING;    (*color name*)
END_VAR
_nColorRGB := nColorRGB;
_sColorName := sColorName;
END_METHOD

METHOD mDisable : BOOL
_bActivate := FALSE;
END_METHOD

METHOD mEnable : BOOL
_bActivate := TRUE;
END_METHOD

{attribute 'monitoring':='call'}
PROPERTY pActive : BOOL
GET
pActive := _bActivate;
END_GET
END_PROPERTY

PROPERTY pErrorCode : INT
GET
pErrorCode := 0;  // no error
END_GET
END_PROPERTY

END_FUNCTION_BLOCK

// ---- POUs/Print/Ads/FB_ADS_CAMERA.TcPOU
FUNCTION_BLOCK FB_ADS_CAMERA EXTENDS FB_AdsBlockBase
VAR
  stAds : ST_ADS_CAMERA;
END_VAR



// Todo redirect PucPath to internal sAdsStruct instead of fb Instance
// - write InstanceName
// - or override getPucPath() (but is PRIVATE)

// The output variables are not used, please add eaccessors if needed
(*
 (*Out*)
  iO_MaxNbMarksQV           : INT := GVL_Camera.cC_QUALIVISION_MAX_NB_MARKS; 
  sO_PointsReadQV           : ST_COMMAND_PLC;    (*New points read by QualiVision*)
  iO_AvailableNbReadPointQV : INT; 
  sO_ReadPointsQV           : ARRAY[1..GVL_Camera.cC_QUALIVISION_MAX_NB_MARKS] OF ST_CAMERA_CORRECTION_QV;
*)

{attribute 'monitoring' := 'call'}
(*
  Name of the block. 
  A friendly name (which is used in the PUC to show the element (only for some blocks/apps))
*)
PROPERTY aName : T_MaxString
GET
aName := aO_Name;
END_GET
SET
aO_Name := aName;
stAds.aO_Name := aName; // update in struct as well
END_SET
END_PROPERTY

PROPERTY bEnable : BOOL
GET
bEnable   := stAds.bI_Enable;   // Set ads interface variable
END_GET
SET
stAds.bI_Enable := bEnable;   // set interface variable
END_SET
END_PROPERTY

METHOD config
VAR_INPUT

END_VAR

//initRemVar();
END_METHOD

PROPERTY eCameraDevice : E_CameraDevice
GET
eCameraDevice := stAds.eI_CameraDevice;
END_GET
SET
stAds.eI_CameraDevice := eCameraDevice;
END_SET
END_PROPERTY

PROPERTY eCameraMode : E_CameraMode
GET
eCameraMode := stAds.eI_CameraMode;
END_GET
SET
stAds.eI_CameraMode := eCameraMode;
END_SET
END_PROPERTY

PROPERTY eTeachProgress : EN_CAMERA_TEACH
GET
eTeachProgress := stAds.eI_TeachProgress;
END_GET
END_PROPERTY

METHOD PROTECTED getPucPath : STRING
VAR
END_VAR
// apply puc path to struct (instead of fb declaraion)
getPucPath := F_Concat3(SUPER^.getPucPath(), '.', 'stAds');
END_METHOD

PROPERTY pCorrectionPointsIndication : POINTER TO ARRAY[1..4] OF ST_CORRECTION_POINT;
GET
pCorrectionPointsIndication := ADR(stAds.sI_CorrectionPointIndication);
END_GET
END_PROPERTY

PROPERTY pTeachPointsQV : POINTER TO ARRAY[1..GVL_Camera.cC_QUALIVISION_MAX_NB_MARKS] OF ST_CAMERA_TEACH_QV;
GET
pTeachPointsQV := ADR(stAds.sI_TeachPointsQV);
END_GET
END_PROPERTY

(*
  Setup constant ADS Block definitions.
  HOWTO: in abstract implmentation call
      init(aVersion:=, aType:=, nType:=, eLayer:=);
*)
METHOD  setup

init(aVersion:=convertVersionIntToString(stAds.iO_Version), aType:=stAds.aO_Type, nType:=ePr_BLK_CAMERA, eLayer:=E_AdsLayer.Structural);
END_METHOD

PROPERTY sMsgInterface : POINTER TO ST_ADS_MSG_IF
GET
sMsgInterface := ADR(stAds.sO_Message);
END_GET
END_PROPERTY

END_FUNCTION_BLOCK

// ---- POUs/Print/Ads/FB_ADS_DVTSHEETALIGNMENT.TcPOU
FUNCTION_BLOCK FB_ADS_DVTSHEETALIGNMENT EXTENDS FB_AdsBlockBase
VAR
  // ---------------------------------
  // ADS interface block specific
  sO_Message         : ST_ADS_MSG_IF;
  
  bI_Enable          : BOOL := TRUE;    (*Enable processing*)

  bI_UsePrintMark    : BOOL := TRUE;    (*Enable processing of print marks*)
  sI_PrintMarkSizeX  : ST_VAR_IN_REAL;  (*Print mark X size [mm]*)
  sI_PrintMarkSizeY  : ST_VAR_IN_REAL;  (*Print mark Y size [mm]*)

  sI_HeadGap         : ST_VAR_IN_REAL;  (*Gap between head and substrate [mm]*)

  lI_SegmentSize     : UDINT;           (*Distance between two images in pixel*)
  lI_SegmentCount    : UDINT;           (*Number of images*)
  fI_SegmentAngle    : REAL;            (*Angle between two segments in deg*)

  sI_DeltaX          : ST_VAR_IN_REAL;  (*X offset between camera marks [mm]*)

  bI_IsMaintenanceJob: BOOL;            (*Maintenance job: disable shift and rotation*)

  (*Out*)
  sO_CurrentAngle    : ST_VAR_OUT_REAL; (*Last measured angle in deg*)
  lO_CurrentYShift   : UDINT;           (*Last measured Y Shift in Pixel*)

  bO_RangeErrorAngle : BOOL;            (*Measured angle out of range*)
  bO_RangeErrorShift : BOOL;            (*Measured shift out of range*)

  // ---------------------------------
END_VAR
VAR PERSISTENT
  aR_Pattern         : UDINT;           (*check pattern for rem validity*)
  bR_Enable          : BOOL;            (*remanent: *)
  bR_UsePrintMark    : BOOL;            (*remanent: *)
  fR_PrintMarkSize_X : REAL;            (*remanent: *)
  fR_PrintMarkSize_Y : REAL;            (*remanent: *)
  fR_HeadGap         : REAL;            (*remanent: head gap in [mm]*)
  fR_DeltaX          : REAL;            (*remanent: *)
END_VAR

PROPERTY bEnable : BOOL
GET
bEnable   := bI_Enable;   // Set ads interface variable
bR_Enable := bI_Enable;   // Update remanent variable
END_GET
SET
bI_Enable := bEnable;   // set interface variable
bR_Enable := bEnable;   // update remanent variable
END_SET
END_PROPERTY

PROPERTY bIsMaintenanceJob : BOOL
GET
bIsMaintenanceJob := bI_IsMaintenanceJob;   // Set ads interface variable
END_GET
SET
bI_IsMaintenanceJob := bIsMaintenanceJob;   // Set ads interface variable
END_SET
END_PROPERTY

PROPERTY bRangeErrorAngle : BOOL
SET
bO_RangeErrorAngle := bRangeErrorAngle;
END_SET
END_PROPERTY

PROPERTY bRangeErrorShift : BOOL
SET
bO_RangeErrorShift := bRangeErrorShift;
END_SET
END_PROPERTY

PROPERTY bUsePrintMark : BOOL
GET
bUsePrintMark   := bI_UsePrintMark;   // Set ads interface variable
bR_UsePrintMark := bI_UsePrintMark;   // Update remanent variable
END_GET
SET
bI_UsePrintMark := bUsePrintMark;   // set interface variable
bR_UsePrintMark := bUsePrintMark;   // update remanent variable
END_SET
END_PROPERTY

METHOD config
VAR_INPUT
  bPrintMarkSizeX_Exist : BOOL;
  aPrintMarkSizeX_Unit  : STRING;
  fPrintMarkSizeX_Min   : REAL;
  fPrintMarkSizeX_Max   : REAL;
  
  bPrintMarkSizeY_Exist : BOOL;
  aPrintMarkSizeY_Unit  : STRING;
  fPrintMarkSizeY_Min   : REAL;
  fPrintMarkSizeY_Max   : REAL;
  
  bHeadGap_Exist        : BOOL;
  aHeadGap_Unit         : STRING;
  fHeadGap_Min          : REAL;
  fHeadGap_Max          : REAL;

  bDeltaX_Exist         : BOOL;
  aDeltaX_Unit          : STRING;
  fDeltaX_Min           : REAL;
  fDeltaX_Max           : REAL;
  
  bCurrentAngle_Exist   : BOOL;
  aCurrentAngle_Unit    : STRING;
  fCurrentAngle_Min     : REAL;
  fCurrentAngle_Max     : REAL;
END_VAR
sI_PrintMarkSizeX.bC_Exist := bPrintMarkSizeX_Exist;
sI_PrintMarkSizeX.aC_Unit  := aPrintMarkSizeX_Unit;
sI_PrintMarkSizeX.fC_Min   := fPrintMarkSizeX_Min;
sI_PrintMarkSizeX.fC_Max   := fPrintMarkSizeX_Max;
sI_PrintMarkSizeY.bC_Exist := bPrintMarkSizeY_Exist;
sI_PrintMarkSizeY.aC_Unit  := aPrintMarkSizeY_Unit;
sI_PrintMarkSizeY.fC_Min   := fPrintMarkSizeY_Min;
sI_PrintMarkSizeY.fC_Max   := fPrintMarkSizeY_Max;
sI_HeadGap.bC_Exist        := bHeadGap_Exist;
sI_HeadGap.aC_Unit         := aHeadGap_Unit;
sI_HeadGap.fC_Min          := fHeadGap_Min;
sI_HeadGap.fC_Max          := fHeadGap_Max;
sI_DeltaX.bC_Exist         := bDeltaX_Exist;
sI_DeltaX.aC_Unit          := aDeltaX_Unit;
sI_DeltaX.fC_Min           := fDeltaX_Min;
sI_DeltaX.fC_Max           := fDeltaX_Max;
sO_CurrentAngle.bC_Exist   := bCurrentAngle_Exist;
sO_CurrentAngle.aC_Unit    := aCurrentAngle_Unit;
sO_CurrentAngle.fC_Min     := fCurrentAngle_Min;
sO_CurrentAngle.fC_Max     := fCurrentAngle_Max;

sO_CurrentAngle.bC_Exist   := FALSE;

initRemVar();
END_METHOD

PROPERTY fDeltaX : REAL
GET
fDeltaX   := sI_DeltaX.fI_Val;   // Set ads interface variable
fR_DeltaX := sI_DeltaX.fI_Val;
END_GET
END_PROPERTY

// HeadGap in [mm]
PROPERTY fHeadGap : LREAL
GET
fHeadGap   := sI_HeadGap.fI_Val;   // Set ads interface variable
fR_HeadGap := sI_HeadGap.fI_Val;   // Update remanent variable
END_GET
SET
sI_HeadGap.fI_Val := TO_REAL(fHeadGap);   // set interface variable
fR_HeadGap        := TO_REAL(fHeadGap);   // update remanent variable
END_SET
END_PROPERTY

PROPERTY fMarkSizeX : REAL
GET
fMarkSizeX         := sI_PrintMarkSizeX.fI_Val;   // Set ads interface variable
fR_PrintMarkSize_X := sI_PrintMarkSizeX.fI_Val;   // Update remanent variable
END_GET
END_PROPERTY

PROPERTY fMarkSizeY : REAL
GET
fMarkSizeY         := sI_PrintMarkSizeY.fI_Val;   // Set ads interface variable
fR_PrintMarkSize_Y := sI_PrintMarkSizeY.fI_Val;   // Update remanent variable
END_GET
END_PROPERTY

PROPERTY fO_CurrentAngle : LREAL
SET
sO_CurrentAngle.fO_Val := tO_REAL(fO_CurrentAngle);
END_SET
END_PROPERTY

PROPERTY fSegmentAngle : REAL
GET
fSegmentAngle := fI_SegmentAngle;   // Set ads interface variable
END_GET
END_PROPERTY

METHOD PROTECTED initRemVar
(*load default initial values if pattern was invalid*)
IF aR_Pattern <> 16#ABCD THEN
  aR_Pattern  := 16#ABCD;  
  bR_Enable   := TRUE;
  bR_UsePrintMark := 0;
  fR_PrintMarkSize_X := 0;
  fR_PrintMarkSize_Y := 0;
  fR_HeadGap  := 2;
  fR_DeltaX := 0;
END_IF

bI_Enable := bR_Enable;
bI_UsePrintMark := bR_UsePrintMark;
sI_PrintMarkSizeX.fI_Val := fR_PrintMarkSize_X;
sI_PrintMarkSizeY.fI_Val := fR_PrintMarkSize_Y;
sI_HeadGap.fI_Val := fR_HeadGap;
sI_DeltaX.fI_Val := fR_DeltaX;
END_METHOD

PROPERTY nO_CurrentYShift : UDINT
SET
lO_CurrentYShift := nO_CurrentYShift;
END_SET
END_PROPERTY

PROPERTY nSegmentCount : UDINT
GET
nSegmentCount := lI_SegmentCount;   // Set ads interface variable
END_GET
END_PROPERTY

PROPERTY nSegmentSize : UDINT
GET
nSegmentSize := lI_SegmentSize;   // Set ads interface variable
END_GET
END_PROPERTY

(*
  Setup constant ADS Block definitions.
  HOWTO: in abstract implmentation call
      init(aVersion:=, aType:=, nType:=, eLayer:=);
*)
METHOD  setup
init(aVersion:='01.00.10', aType:='DvtSheetAlignment', nType:=ePr_BLK_SA, eLayer:=E_AdsLayer.Structural);
END_METHOD

PROPERTY sMsgInterface : POINTER TO ST_ADS_MSG_IF
GET
sMsgInterface := ADR(sO_Message);
END_GET
END_PROPERTY

END_FUNCTION_BLOCK

// ---- POUs/Print/Camera/FB_CameraBase.TcPOU
(*
  Base camera system
  Implements I_Camera: set I_CameraSink.   
*)
FUNCTION_BLOCK ABSTRACT FB_CameraBase EXTENDS FB_Commons IMPLEMENTS I_Camera, I_CameraTriggerDevice

VAR
  _bInitialized             : BOOL;
  _iCameraSink              : I_CameraSink;
  _iCameraTrigger           : I_CameraTrigger;
  _bSimulate                : BOOL;
  _nPrintUnitResolution     : UDINT;           (*printhead pixel resolution [dpi]*)
  _nPrintUnitSubPx          : UDINT;           (*print unit SubPixel resolution [SubPx]*)
  _bUseCameraTrigger        : BOOL;            (*use a trigger output timestamp I/O*)
  _bUseCameraTriggerFeedback : BOOL;           (*use a camera triggered feedback timestamp I/O*)
  _eCameraMode              : E_CameraMode;    (*desired camera mode*)
  _ePossibleMode            : E_CameraMode;    (*currently possible mode*)
  _fSubstrateLength         : LREAL := 1;      (*Substrate length [m]*)
  _fSubstrateWidth          : LREAL := 1;      (*Substrate width [m]*)
  _fImageLength             : LREAL := 1;      (*Image length [m]*)
  _fImageWidth              : LREAL := 1;      (*Image width [m]*)
  _fFrameLength             : LREAL := 1;      (*Camera Frame width in [px]*)
  _bActivated               : BOOL;            (*Camera is activated*)
  _sVisuName                : STRING := 'unvailable';     (*detail visualisation instance name*)
  
  // status
  _bCamTriggerOk            : BOOL;
  _bCamTriggerStarted       : BOOL;
  _bCamTriggerDone          : BOOL;   
  _nCamStartPos             : DINT;            (*Cam start position ideal [SubPx]*)
  _nCamStartPosDeviation    : DINT;            (*Cam stated position real [SubPx]*)
  _nRxCamPoints             : UDINT;           (*number of received cam points*)

  // helper
  stCamPoint                : ST_DeformationPointAccurate;(*actual camera point*)
    
  // messaging
  _pMsgConfig               : POINTER TO CalmarCommons.ST_MSG_CONFIG;
END_VAR

VAR PERSISTENT
  _fTriggerDistance         : LREAL;           (*[m] Distance between Sensor and Trigger*)
  _fTriggerPulseLength      : LREAL := 10;     (*[ms] Length of trigger signal in ms, min. 3 bus cycles*)
  _fDetectToCameraOffset    : LREAL := 0.1;    (*[m] Distance between input trigger and camera, mech.*)
  _fCameraToPrintOffset     : LREAL := 0.0;    (*[m] Distance between Camera and PU, mech, This offset can be used to shift the reference of a camera/sheet-detect, e.g. because this reference is different from to one where the alignment Camera/sheetdetect-PrintUnit has been made*)
END_VAR

METHOD ActivateCam : BOOL
VAR_INPUT
  iCameraSink : I_CameraSink;
END_VAR
IF iCameraSink = 0 THEN
  LogError('Invalid parameter (0 pointer)');
  ActivateCam := FALSE;
  RETURN; 
ELSIF _iCameraSink <> 0 AND iCameraSink <>_iCameraSink THEN
  LogError('SetSink failed: other sink already exists');
  ActivateCam := FALSE;
  RETURN; 
END_IF 

_iCameraSink := iCameraSink;
_iCameraTrigger.Enable(iCam:=THIS^, bUseCameraTrigger:=_bUseCameraTrigger, bUseCameraTriggerFeedback:=_bUseCameraTriggerFeedback);

_bActivated := TRUE;
ActivateCam:=TRUE;
END_METHOD

(*
  Activate/Deactivate camera trigger device
*)
PROPERTY bEnableTrigger : BOOL
SET
IF bEnableTrigger THEN
  _iCameraTrigger.Enable(iCam := THIS^, bUseCameraTrigger:= _bUseCameraTrigger, bUseCameraTriggerFeedback:=_bUseCameraTriggerFeedback);
ELSE
  _iCameraTrigger.Disable();
END_IF
END_SET
END_PROPERTY

(*
  Activate/Deactivate camera manual teach mode
*)
PROPERTY bManualTeach : BOOL
SET
_iCameraTrigger.bManualTeach := bManualTeach;
END_SET
END_PROPERTY

{attribute 'monitoring':='call'}
PROPERTY bSimulate : BOOL
GET
bSimulate := _bSimulate;
END_GET
SET
_bSimulate := bSimulate;
END_SET
END_PROPERTY

METHOD CamTrigger
VAR_INPUT
  bOk             : BOOL;     // trigger is ok
	nPos            : DINT;     // camera triggered position
  nPosDeviation   : DINT;     // camera started deviation
  nX0             : DINT;     // detected position sheet/repetition
END_VAR
_nRxCamPoints := 0;
_bCamTriggerStarted    := TRUE;
_bCamTriggerDone       := FALSE;
_bCamTriggerOk  := bOk;
_nCamStartPos   := nPos;
_nCamStartPosDeviation := nPosDeviation;

LogLvl(Lvl:=E_LogSeverity.Debug, Msg:=F_Concat2('CamTrigger at X0=', TO_STRING(nPos)));
IF _iCameraSink <> 0 THEN   // inform sink
  _iCameraSink.CamStarted(nX0:=nX0);
END_IF
END_METHOD

METHOD CamTriggerDone
_bCamTriggerStarted    := FALSE;  // this call marks the end of the camera trigger period
_bCamTriggerDone       := TRUE;

LogLvl(Lvl:=E_LogSeverity.Debug, Msg:='CamTriggerDone');
IF _iCameraSink <> 0 THEN   // inform sink
  _iCameraSink.CamDone();
END_IF
END_METHOD

METHOD DeactivateCam : BOOL
VAR_INPUT
  iSink : I_CameraSink;
END_VAR
IF _iCameraSink <> 0 AND iSink <> _iCameraSink THEN
  LogError('remove sink failed: inconsistent');
  DeactivateCam := FALSE;
  RETURN;  
END_IF

_iCameraSink := 0;
_iCameraTrigger.Disable();
_bActivated := FALSE;
DeactivateCam:=TRUE;
END_METHOD

{attribute 'monitoring':='call'}
PROPERTY ABSTRACT eCameraMode : E_CameraMode
GET
END_GET
END_PROPERTY

{attribute 'monitoring':='call'}
PROPERTY ABSTRACT eDeviceType : E_CameraDevice
GET
END_GET
END_PROPERTY

{attribute 'monitoring':='call'}
PROPERTY fCameraToPrintOffset : LREAL
GET
//This offset can be used to shift the reference of a camera, e.g. because this reference is different from to one where the alignment Camera-PrintUnit has been made
fCameraToPrintOffset := _fCameraToPrintOffset;
END_GET
SET
_fCameraToPrintOffset := fCameraToPrintOffset;
END_SET
END_PROPERTY

{attribute 'monitoring':='call'}
PROPERTY fDetectToCameraOffset : LREAL
GET
//This offset can be used to shift the reference of a camera, e.g. because this reference is different from to one where the alignment Camera-PrintUnit has been made
fDetectToCameraOffset := _fDetectToCameraOffset;
END_GET
SET
_fDetectToCameraOffset := fDetectToCameraOffset;
END_SET
END_PROPERTY

{attribute 'monitoring':='call'}
(* camera frame size in [px]*)
PROPERTY fFrameLength : LREAL
GET
fFrameLength := _fFrameLength;
END_GET
SET
_fFrameLength := fFrameLength;
END_SET
END_PROPERTY

{attribute 'monitoring':='call'}
(*Image Length/Depth in [m]*)
PROPERTY fImageLength : LREAL
GET
fImageLength := _fImageLength;
END_GET
SET
_fImageLength := fImageLength;
END_SET
END_PROPERTY

{attribute 'monitoring':='call'}
(*Image Width in [m]*)
PROPERTY fImageWidth : LREAL
GET
fImageWidth := _fImageWidth;
END_GET
SET
_fImageWidth := fImageWidth;
END_SET
END_PROPERTY

{attribute 'monitoring':='call'}
(*Substrate Length/Depth in [m]*)
PROPERTY fSubstrateLength : LREAL
GET
fSubstrateLength := _fSubstrateLength;
END_GET
SET
//ROI in Print direction
IF _iCameraTrigger <> 0 THEN
  _iCameraTrigger.SetSubstrateLength(fSubstrateLength := fSubstrateLength);   // save to camera trigger
  _fSubstrateLength := fSubstrateLength;                                      // save to camera
END_IF
END_SET
END_PROPERTY

{attribute 'monitoring':='call'}
(*Substrate Width in [m]*)
PROPERTY fSubstrateWidth : LREAL
GET
fSubstrateWidth := _fSubstrateWidth;
END_GET
SET
_fSubstrateWidth := fSubstrateWidth;
END_SET
END_PROPERTY

{attribute 'monitoring':='call'}
PROPERTY fTriggerDistance : LREAL
GET
fTriggerDistance := _fTriggerDistance;
END_GET
SET
_fTriggerDistance := fTriggerDistance;
END_SET
END_PROPERTY

PROPERTY fTriggerPulseLength : LREAL
GET
fTriggerPulseLength := _fTriggerPulseLength;
END_GET
END_PROPERTY

METHOD ABSTRACT GetCamStatus : BOOL
VAR_OUTPUT
  bConnectionOK  : BOOL;    // Camera connected
  bTeachOk       : BOOL;    // Teach successful
  nTeachedPoints : UDINT;   // Teached points for this job
  nScannedPoints : UDINT;   // Scanned points on current sheet  
  bCamStarted    : BOOL;    // Camera trigger is active, cam started
  bCamDone       : BOOL;    // Camera finished on last CT
  bErrors        : ARRAY[1..GVL_Camera.nC_NbCamErrors] OF BOOL;  // generic error flag list
END_VAR
END_METHOD

METHOD Init
VAR_INPUT
  nPrintUnitResolution         : UDINT;    (*printhead pixel resolution [dpi]*)
  nPrintUnitSubPx              : UDINT;    (*print unit subPixel resolution [SubPx]*)
  iCameraTrigger               : I_CameraTrigger;
  bUseCameraTrigger            : BOOL;     (*use a trigger output timestamp I/O*)
  bUseCameraTriggerFeedback    : BOOL;     (*use a camera triggered feedback timestamp I/O*)
END_VAR
IF nPrintUnitResolution <> 0 AND iCameraTrigger <> 0 THEN
  _nPrintUnitResolution := nPrintUnitResolution;
  _nPrintUnitSubPx      := nPrintUnitSubPx;
  _iCameraTrigger       := iCameraTrigger;
  
  _bUseCameraTrigger := bUseCameraTrigger;
  _bUseCameraTriggerFeedback := bUseCameraTriggerFeedback;
  
  _bInitialized := TRUE;
ELSE
  _bInitialized := FALSE;
END_IF
END_METHOD

METHOD mJobStart : BOOL
END_METHOD

(*
  Set mode to camera.
  :return: TRUE if success
*)
METHOD ABSTRACT setCameraMode : BOOL
VAR_INPUT
  eCameraMode : E_CameraMode;
END_VAR
END_METHOD

METHOD setMsgInterface : BOOL
VAR_INPUT
	pMsgConfig	: POINTER TO CalmarCommons.ST_MSG_CONFIG;
END_VAR
_pMsgConfig := pMsgConfig;
END_METHOD

{attribute 'monitoring':='call'}
PROPERTY sName : STRING
GET
sName := 'undefined';
END_GET
END_PROPERTY

{attribute 'monitoring':='call'}
PROPERTY sVisuName : STRING
GET
sVisuName := _sVisuName;
END_GET
SET
_sVisuName := sVisuName;
END_SET
END_PROPERTY

END_FUNCTION_BLOCK

// ---- POUs/Print/Camera/FB_CameraDummy.TcPOU
FUNCTION_BLOCK FB_CameraDummy EXTENDS FB_CameraBase
VAR_INPUT
END_VAR
VAR_OUTPUT
END_VAR
VAR
END_VAR

{attribute 'monitoring':='call'}
PROPERTY eCameraMode : E_CameraMode
GET
eCameraMode := _eCameraMode;
IF _eCameraMode = E_CameraMode.Auto THEN
  eCameraMode := E_CameraMode.NoCorrection;
END_IF
END_GET
END_PROPERTY

PROPERTY eDeviceType : E_CameraDevice
GET
eDeviceType := E_CameraDevice.SheetDetect;
END_GET
END_PROPERTY

METHOD GetCamStatus : BOOL
VAR_OUTPUT
  bConnectionOK  : BOOL;    // Camera connected
  bTeachOk       : BOOL;    // Teach successful
  nTeachedPoints : UDINT;   // Teached points for this job
  nScannedPoints : UDINT;   // Scanned points on current sheet
  bCamStarted    : BOOL;    // Camera trigger is active, cam started
  bCamDone       : BOOL;    // Camera finished on last CT
  bErrors        : ARRAY[1..GVL_Camera.nC_NbCamErrors] OF BOOL;  // generic error flag list
END_VAR
bConnectionOK  := TRUE;  //NO comm with a cam 
bTeachOk       := TRUE;  //NO teach availabe
nTeachedPoints := 0;
nScannedPoints := 0;
bCamStarted    := _bCamTriggerStarted;
bCamDone       := _bCamTriggerDone;

GetCamStatus := TRUE;
END_METHOD

(*
  Set mode to camera.
  :return: TRUE if success
*)
METHOD setCameraMode : BOOL
VAR_INPUT
  eCameraMode : E_CameraMode;
END_VAR
IF eCameraMode = E_CameraMode.NoCorrection THEN   // supported mode
  
  _eCameraMode := eCameraMode; 
  setCameraMode := TRUE;        // set desired mode
ELSE
  LogError(F_Concat3('Camera mode=', TO_STRING(eCameraMode), ' not supported by camera'));
  _eCameraMode := E_CameraMode.NoCorrection;
END_IF
END_METHOD

{attribute 'monitoring':='variable'}
PROPERTY sName : STRING
GET
sName := 'SheetDetect';
END_GET
END_PROPERTY

END_FUNCTION_BLOCK

// ---- POUs/Print/Camera/FB_CameraTcpIp.TcPOU
(*
  Base camera system with TcpIp communicatiom
  Implements callback function (rx_callback) for received TcpIp messages.   
*)
FUNCTION_BLOCK ABSTRACT FB_CameraTcpIp EXTENDS FB_CameraBase IMPLEMENTS I_TcpIp_RxMsgHandler

VAR
  sLastMessage              : STRING(GVL_TcpIp.TCP_RXDATA_SIZE);          (*rx telegram string*)
  nLastMessageSz            : UDINT;                                      (*receive message length *)
  sMemLastMessage           : STRING(GVL_TcpIp.TCP_RXDATA_SIZE);          (*mem rx telegram string*)
  nRxMsg                    : UDINT;                (*rx telegram counter*)
  bMsgReceived              : BOOL;                 (*we received a message*)
  sState                    : STRING;               (*state change event as string*)

  sLastErrorMessage         : STRING(GVL_TcpIp.TCP_RXDATA_SIZE);          (*rx telegram error string*)
  _bConnectionError         : BOOL;
  _pFbTcpIpClient           : POINTER TO FB_TcpClient;
END_VAR

METHOD ActivateCam : BOOL
VAR_INPUT
  iCameraSink : I_CameraSink;
END_VAR
ActivateCam := SUPER^.ActivateCam(iCameraSink:=iCameraSink);

IF _pFbTcpIpClient = 0 THEN
  LogError('No tcpip client assigned');
  ActivateCam := 0;
  RETURN;
END_IF

_pFbTcpIpClient^.bEnable := TRUE;
END_METHOD

PROPERTY bConnectionErr : BOOL
GET
IF _pFbTcpIpClient = 0 THEN RETURN; END_IF

_bConnectionError := FALSE;
IF _bActivated THEN
  IF NOT _pFbTcpIpClient^.bConnected OR _pFbTcpIpClient^.bError THEN
    bConnectionErr := TRUE;
    _bConnectionError := TRUE;
  END_IF 
END_IF
END_GET
END_PROPERTY

METHOD DeactivateCam : BOOL
VAR_INPUT
  iSink : I_CameraSink;
END_VAR
DeactivateCam := SUPER^.DeactivateCam(iSink:=iSink);

IF _pFbTcpIpClient = 0 THEN
  LogError('No tcpip client assigned');
  DeactivateCam := 0;
  RETURN;
END_IF

_pFbTcpIpClient^.bEnable := FALSE;
END_METHOD

METHOD ABSTRACT GetCamStatus : BOOL
VAR_OUTPUT
  bConnectionOK  : BOOL;    // Camera connected
  bTeachOk       : BOOL;    // Teach successful
  nTeachedPoints : UDINT;   // Teached points for this job
  nScannedPoints : UDINT;   // Scanned points on current sheet
  bCamStarted    : BOOL;    // Camera trigger is active, cam started
  bCamDone       : BOOL;    // Camera finished on last CT
  bErrors        : ARRAY[1..GVL_Camera.nC_NbCamErrors] OF BOOL;  // generic error flag list
END_VAR
END_METHOD

METHOD rx_callback
VAR_INPUT
	sMessage	: CalmarCompTcpIp.ST_TcpMsg;
END_VAR
sLastMessage  := sMessage.sMessage;   // store message locally
nRxMsg        := nRxMsg + 1;
nLastMessageSz := LEN2(ADR(sLastMessage));

bMsgReceived  := TRUE;
END_METHOD

METHOD setTcpIpClient : BOOL
VAR_INPUT
  pTcpIpClient  : POINTER TO FB_TcpClient;
END_VAR
_pFbTcpIpClient := pTcpIpClient;
END_METHOD

METHOD state_callback
VAR_INPUT
	(* state change event as string (think to convert it to an enum for easier handling later)*)
	state	: STRING;
END_VAR
sState := state;   // store state locally
END_METHOD

END_FUNCTION_BLOCK

// ---- POUs/Print/Camera/FB_CameraTrigger.TcPOU
FUNCTION_BLOCK FB_CameraTrigger EXTENDS FB_Commons IMPLEMENTS I_CameraTrigger, I_StartPosDetect
(*************************************************************************************************)
(*  FILENAME:    FB_CameraTrigger                                                                *)
(*  PROJECT:     CALMAR PUPLC                                                                    *)
(*  COPYRIGHT:   All rights reserved (c) Wifag//Polytype, Fribourg/Switzerland (2016)            *)
(*  ENVIRONMENT: TwinCAT PLC                                                                     *)
(*  VERSION:     <version>                                                                       *)
(*************************************************************************************************)
(*  DESCRIPTION:                                                                   <description> *)
(*    Generate timestamp trigger output based on timestamp sensor input. Two variants            *)
(*    exist, a timebased approach where the trigger time is calculated at the time the sensor    *)
(*    event occurs, and a second approach where the sensor event time is translated to a sensor  *)
(*    event position, and a trigger is generated when the calculated trigger position has almost *)
(*    been reached. The second approach has the advantage that is is less susceptible to speed   *)
(*    variations.                                                                                *)
(*                                                                                </description> *)
(*************************************************************************************************)

{library public}
VAR_INPUT
  bI_HwEnable                             : BOOL;            // relase (enable SheetDetect) from machine
  bI_AutomaticMode                        : BOOL;            // machine is in automatic mode
  (* - (EL1252) StartPosition detect sensor*)
  bI_SensorSupervisionEnable              : BOOL := TRUE;    // enable SheetDetect with supervision 
  bI_Sensor_State                   AT%I* : BOOL;            // Sensor signal
  tI_Sensor_TimeStampPos            AT%I* : T_DCTIME64;      // Sensor last detection timestamp
  (* - (EL1252) Camera started feedback trigger/signal*)
  bI_TriggerFeedback_State          AT%I* : BOOL;           // Sensor signal
  tI_TriggerFeedback_TimeStampPos   AT%I* : T_DCTIME64;     // Sensor last detection timestamp

  (*System signals*)
  iI_CurrentPos                   : DINT;                   // Current position in [SubPx]*)
  fI_ConveyorSpeed                : LREAL;                  // Current speed of substrate in [m/s]*)
  
  (*Debug & Test*)
  bI_ManualTrigger                : BOOL;                   // Manual start trigger
END_VAR

VAR_OUTPUT
  (*Link to EL2252*)
  ObTrigger                 AT%Q* : BOOL;                   // EL2252 Output1 - TRUE=start camer
  OtTriggerStartTime        AT%Q* : T_DCTIME64;             // EL2252 Timestamp - where to set outputs
  OnTriggerCommand          AT%Q* : BYTE;                   // EL2252 Command - activation timestamp ouput
END_VAR

(*{library private}*)
VAR
  bInitOk                         : BOOL;           // initialized
  bSpeedValid                     : BOOL;           // speed is valid
  bTriggerEnabled                 : BOOL;           // detection & trigger is enabled
  bTriggerArmed                   : BOOL;           // trigger is armed
  bCamValid                       : BOOL;           // camera is valid
  bTriggerOk                      : BOOL;
  rT_Sensor                       : R_TRIG;        // rising edge trigger sensor
  
  (*configuration*)
  _nResolution                    : INT := 1;       // Printhead Resolution [e.g. 600] x Subpixel Resolution [e.g. 32]*)
  _bUsePositionTrigger            : BOOL;           // FALSE: Calculate time with speed and position distance@sensor event, TRUE: Calculate sensor event position, launch trigger based on position
  _bUseCameraTrigger              : BOOL;           // (cam specific setting) Generate camera trigger output
  _bUseCameraTriggerFeedback      : BOOL;           // (cam specific setting) Evaluate camera triggered feedback
  _bCamManualTeachMode            : BOOL;           // cam in manual teach mode
  _tMemTriggerFeedback_TimeStampPos : T_DCTIME64;
  _nSubstrateLength               : DINT;           // Substrate length in pulse [SubPx]
  _fSubstrateLength               : LREAL;          // Substrate length in [m]
  _fTriggerDistance               : LREAL;          // Distance between Sensor and Trigger [m]
  _fTriggerLength                 : LREAL := 10;    // Length of trigger signal in ms, min. 3 bus cycles
  
  iActiveCam	                    : I_CameraTriggerDevice;  // active camera interface
  
  bSheetDetected                  : BOOL;
  bInhibitTrigger                 : BOOL;            (*inhibit trigger signals, TRUE=inhibit*)
  bReleaseInhibitTrigger          : BOOL;            (*condition to release inhibit trigger*)

  eState                          : BYTE;            (*State*)
  tSensor_TimeStamp               : T_DCTIME64;      (*Sensor last detection timestamp*)
  tTriggerFeedback_TimeStamp      : T_DCTIME64;      (*Trigger feedback last detection timestamp*)
  tCurrentTime                    : T_DCTIME64;      (*Current system dc time [64bit]*)
  tTrigger_EventTime              : T_DCTIME64;      (*Trigger event timestamp*)

  _bManualStart                   : BOOL;
  fDeltaDistance                  : LREAL;           (*Distance that the substrate moved between the detection and the treatment of the information [m]*)
  _nX0                            : DINT;            (*Detected X0 position of CT [SubPx] by sensor*)
  _nCamStartPos                   : DINT;            (*Camera start position*)
  _nCamStartedPos                 : DINT;            (*Camera started position [SubPx]*)
  
  tCurrentTimeStamp               : T_DCTIME64;      (* Get Current Timestamp *)
  tLastTimeStamp                  : T_DCTIME64;      (* Get Current Timestamp *)
  fCycleTime                      : LREAL;           (* Current calculated cycle time [s]*)

  fRemDist                        : LREAL;           (*Remaining distance until trigger occurs [m]*)
  fPreTriggerPosition             : LREAL;           (*Margin between effective trigger position and generation of timestamp*)

  (*Debug*)
  _bVerbose                       : BOOL;
END_VAR

VAR CONSTANT
  fC_MIN_CONVEYOR_SPEED           : LREAL := 0.01;
  fC_PreTrigFactor                : LREAL := 3.0;
  fC_SheetLengthMargin            : LREAL := 0.01;   (*Added 10 mm margin for substrate length in case of print quality strips at the end of sheet in case of start with edge*)
  fC_MaxCameraFeedbackTimeout     : LREAL := 28.0;   (*[ns] Max. timeout waiting for camera trigger feedback signal*)

  (*State*)
  cL_IDLE                         : BYTE := 0;       (*Idle state, no trigger active*)
  cL_SENSOREVENT                  : BYTE := 1;       (*Sensor started trigger generation*)
  cL_WAITALMOSTSTART              : BYTE := 2;       (*Wait timestamp calculation critera*)
  cL_WAITSTART                    : BYTE := 3;       (*Wait for trigger generation critera*)
  cL_WAITFEEDBACK                 : BYTE := 4;       (*Wait on feedback from trigger*)
  cL_TRIGACTIVE                   : BYTE := 5;       (*Trigger set*)
  cL_WAITSTOP                     : BYTE := 6;       (*Trigger reset*)

  (*EL2252 Command*)
  nC_EL2252Cmd_INACTIVE           : BYTE := 0;
  nC_EL2252Cmd_ACTIVE             : BYTE := 3;
END_VAR

IF NOT bInitOk THEN RETURN; END_IF;

// General calculations
bSpeedValid   := fI_ConveyorSpeed > fC_MIN_CONVEYOR_SPEED;    // speed valid (ignore trigger if not moving)
bCamValid     := SEL(iActiveCam<>0, FALSE, TRUE);             // camera valid (ignore trigger otherwise)
tCurrentTime  := F_GetCurDcTaskTime64();                      // current dc time (most accurate time stamp we have)
fCycleTime    := (TO_LREAL(tCurrentTime) - TO_LREAL(tLastTimeStamp)) * 1E-9;  tLastTimeStamp  := tCurrentTime;  // calculate cycle time of this block
bSheetDetected:= FALSE;                                       // Set to true below just for one cycle
bTriggerEnabled := bSpeedValid AND bI_HwEnable AND (bI_AutomaticMode OR _bCamManualTeachMode);
bTriggerArmed :=  NOT bInhibitTrigger AND bTriggerEnabled;
rT_Sensor(CLK := bI_Sensor_State AND bI_SensorSupervisionEnable);

// apply parameter
IF bCamValid THEN    // save dynamic changable settings
  _fTriggerDistance := iActiveCam.fTriggerDistance;
  _fTriggerLength   := iActiveCam.fTriggerPulseLength;
END_IF

// - Release inhibit trigger
bReleaseInhibitTrigger := bInhibitTrigger AND (iI_CurrentPos - (_nX0 + _nSubstrateLength)) > 0;
IF bReleaseInhibitTrigger THEN bInhibitTrigger := FALSE; END_IF

// Reset trigger if deactivated - should improve hanging triggers
IF NOT bTriggerEnabled AND eState > cL_IDLE THEN
  Reset();
  RETURN;
END_IF


(*State Machine ----------------------------------------------------------------*)
CASE eState OF
  cL_IDLE:     (*Not started, waiting for start trigger*)
  
    IF bTriggerArmed THEN (*ignore trigger else*)
 
      IF rT_Sensor.Q AND (bCamValid OR _bCamManualTeachMode) THEN      (*Start launched*)
        eState            := cL_SENSOREVENT;
        tSensor_TimeStamp := tI_Sensor_TimeStampPos;
        _bManualStart := FALSE;
        IF _bCamManualTeachMode THEN LogWarning('StartTrigger in manual teach mode'); END_IF
      ELSIF (bI_ManualTrigger AND bCamValid) THEN  (*Manual start launched*)
        eState            := cL_SENSOREVENT;
        tSensor_TimeStamp := tCurrentTime;
        _bManualStart := TRUE;
      ELSIF (rT_Sensor.Q OR bI_ManualTrigger) AND NOT bCamValid THEN   (*Trigger without active camera*)
        LogWarning('No camera or start device active, ignore trigger');
      END_IF;
      
    END_IF
    
    OnTriggerCommand := nC_EL2252Cmd_INACTIVE;
    ObTrigger        := FALSE;

  cL_SENSOREVENT:     (*Not started*)
    IF NOT bSpeedValid THEN 
      Reset();        // ignore trigger if not moving anymore (avoid zero division)
    ELSE
      (*Distance in [m] that the substrate has traveled between the sensor detection (time) current plc cycle*)
      fDeltaDistance     := UINT64_TO_LREAL(UInt64Sub64(ULINT_TO_ULARGE(tCurrentTime), ULINT_TO_ULARGE(tSensor_TimeStamp))) * 1E-9 * fI_ConveyorSpeed;
      (*Position where the sheet has been detected in [SubPx]*)
      _nX0               := iI_CurrentPos - F_MeterToSubPixel(fPosMeter:=fDeltaDistance, fResoSubPx:=_nResolution);
      
      IF _bUsePositionTrigger OR NOT _bUseCameraTrigger THEN
        eState             := cL_WAITALMOSTSTART;
      ELSE
        eState             := cL_WAITSTART;
        tTrigger_EventTime := (tSensor_TimeStamp + LREAL_TO_ULINT(_fTriggerDistance / fI_ConveyorSpeed * 1E9));
      END_IF;
      
      OnTriggerCommand := nC_EL2252Cmd_INACTIVE;
      ObTrigger         := TRUE;
      bInhibitTrigger   := TRUE;
      bSheetDetected    := TRUE;
      
    END_IF

  cL_WAITALMOSTSTART: (*Only active when bI_UsePositionTrigger=TRUE: wait until Start position almost reached, then set timestamp*)
    (*Remaining distance in [m], converted to REAL to avoid integer wrap problems*)
    fRemDist             := _fTriggerDistance + (DINT_TO_REAL(_nX0) - DINT_TO_REAL(iI_CurrentPos))*0.0254 / INT_TO_REAL(_nResolution);
    fPreTriggerPosition  := fC_PreTrigFactor * fCycleTime * fI_ConveyorSpeed;

    IF fRemDist < fPreTriggerPosition THEN
      eState             := cL_WAITSTART;
      tTrigger_EventTime := (tSensor_TimeStamp + LREAL_TO_ULINT(fRemDist / fI_ConveyorSpeed * 1E9));    // division save because we are moving to reach this position
      IF _bUseCameraTrigger AND NOT _bManualStart THEN
        OnTriggerCommand := nC_EL2252Cmd_ACTIVE;  (*Arm EL2252*)
      END_IF
      LogTsDiff(aIdent:= 'WAITALMOSTSTART: ', t1:=tTrigger_EventTime, t2:=tCurrentTime);
    ELSE
      eState           := cL_WAITALMOSTSTART;
      OnTriggerCommand := nC_EL2252Cmd_INACTIVE;
    END_IF;
    ObTrigger          := TRUE;

  cL_WAITSTART:       (*Wait until start time reached*)
    bTriggerOk := TRUE;
    IF (tTrigger_EventTime < tCurrentTime) THEN (* StartTime elapsed *)
      // position reached
      IF _bUseCameraTriggerFeedback THEN
        eState         := cL_WAITFEEDBACK;
      ELSE
        eState         := cL_TRIGACTIVE;
        iActiveCam.CamTrigger(bOk:=bTriggerOk, nPos:=iI_CurrentPos, nPosDeviation:=0, nX0:=_nX0);
      END_IF

      OnTriggerCommand := nC_EL2252Cmd_INACTIVE; (*Disarm already command to EL2252, trigger generated*)
    ELSE
      // position not yet reached
      eState           := cL_WAITSTART;
      IF _bUseCameraTrigger AND NOT _bManualStart THEN
        OnTriggerCommand := nC_EL2252Cmd_ACTIVE;  (*Arm EL2252*)
      END_IF
    END_IF;

    ObTrigger      := TRUE;  
    
  cL_WAITFEEDBACK:
    IF _bManualStart THEN //Simulate feedback in case of manual start
      tTriggerFeedback_TimeStamp:= tTrigger_EventTime + LREAL_TO_ULINT(1000.0 * 1E3); //Trigger event plus 1000ns
    ELSE
      IF tI_TriggerFeedback_TimeStampPos = _tMemTriggerFeedback_TimeStampPos AND tCurrentTime > (tTrigger_EventTime + LREAL_TO_ULINT(fC_MaxCameraFeedbackTimeout * 1E3)) THEN
        // feedback was not received in next plc cycle (timeout jitter in camera max. 28us)
        LogError(F_Concat3('No Camera trigger feedback received (timeout), after ', TO_STRING(TO_LREAL(tCurrentTime-tTrigger_EventTime)/1E6), 'ms'));
        bTriggerOk := FALSE;
        tTriggerFeedback_TimeStamp:= tTrigger_EventTime + LREAL_TO_ULINT(fC_MaxCameraFeedbackTimeout * 1E3);
      ELSE
        tTriggerFeedback_TimeStamp:= tI_TriggerFeedback_TimeStampPos;
			END_IF
    END_IF
    
  (*feedback signal is a very short trigger that the PLC sometimes cannot register, therefore we use the timestamp*)
    IF (tTriggerFeedback_TimeStamp <> _tMemTriggerFeedback_TimeStampPos) AND (tTriggerFeedback_TimeStamp > 0) OR _bManualStart THEN
      eState          := cL_TRIGACTIVE;
      // start position requested
      fDeltaDistance  := UINT64_TO_LREAL(UInt64Sub64(ULINT_TO_ULARGE(tCurrentTime), ULINT_TO_ULARGE(tTrigger_EventTime))) * 1E-9 * fI_ConveyorSpeed;
      _nCamStartPos   := _nX0 +   F_MeterToSubPixel(fPosMeter:=_fTriggerDistance, fResoSubPx:=_nResolution);
      
      // effective started position
      fDeltaDistance  := UINT64_TO_LREAL(UInt64Sub64(ULINT_TO_ULARGE(tCurrentTime), ULINT_TO_ULARGE(tTriggerFeedback_TimeStamp))) * 1E-9 * fI_ConveyorSpeed;
      _nCamStartedPos := iI_CurrentPos - F_MeterToSubPixel(fPosMeter:=fDeltaDistance, fResoSubPx:=_nResolution);
      IF _bManualStart THEN iActiveCam.CamTrigger(bOk:=bTriggerOk, nPos:=_nCamStartPos, nPosDeviation:=0, nX0:=_nX0);
      ELSE                  iActiveCam.CamTrigger(bOk:=bTriggerOk, nPos:=_nCamStartPos, nPosDeviation:=-_nCamStartedPos+_nCamStartPos, nX0:=_nX0); END_IF  (*!!!!   sign inverted*)
    ELSE
     eState           := cL_WAITFEEDBACK;
    END_IF    
    
  cL_TRIGACTIVE:   (*Trigger high*)
    eState         := cL_WAITSTOP;
    
    // calculate end timestamp of trigger (end of trigger active signal)
    tTrigger_EventTime := (tTrigger_EventTime + LREAL_TO_ULINT(_fTriggerLength * 1E6));
     
    OnTriggerCommand := nC_EL2252Cmd_INACTIVE;
    ObTrigger        := FALSE;
    
  cL_WAITSTOP:  (*Wait until trigger time has elapsed*)
    IF (tTrigger_EventTime < tCurrentTime) THEN (* StopTime elapsed *)
      eState           := cL_IDLE;
      OnTriggerCommand := nC_EL2252Cmd_INACTIVE; (*Disarm EL2252, trigger generated*)
      iActiveCam.CamTriggerDone();
    ELSE
      eState           := cL_WAITSTOP;
      IF _bUseCameraTrigger THEN
        OnTriggerCommand := nC_EL2252Cmd_ACTIVE;  (*Arm EL2252*)
      END_IF
    END_IF;

    ObTrigger        := FALSE;

  ELSE  (*Default*)
    eState           := cL_IDLE;
    ObTrigger        := FALSE;
    OnTriggerCommand := nC_EL2252Cmd_INACTIVE;
END_CASE;

OtTriggerStartTime := tTrigger_EventTime;  // set output

_tMemTriggerFeedback_TimeStampPos := tI_TriggerFeedback_TimeStampPos;

PROPERTY bManualTeach : BOOL
GET
bManualTeach := _bCamManualTeachMode;
END_GET
SET
_bCamManualTeachMode := bManualTeach;
END_SET
END_PROPERTY

(*
  A new container detected on X0.
  NOTE: a pulse only
*)
PROPERTY bStartTrig : BOOL
GET
bStartTrig := bSheetDetected;
END_GET
END_PROPERTY

(*
  A valid container detected.
*)
PROPERTY bValid : BOOL
GET
bValid := bSheetDetected AND NOT _bCamManualTeachMode AND bCamValid;  // in manual teach the ct is "present" should not be printed
END_GET
END_PROPERTY

METHOD Disable : BOOL
IF eState = cL_IDLE THEN
  iActiveCam := 0;
  Disable := TRUE;
ELSE  
  Disable := FALSE;
  LogError('disable failed: trigger busy -> reset trigger');
  Reset();
END_IF
END_METHOD

METHOD Enable : BOOL
VAR_INPUT
	iCam	                    : I_CameraTriggerDevice;
  bUseCameraTrigger         : BOOL; //Generate camera trigger
  bUseCameraTriggerFeedback : BOOL; //Use feedback as trigger?
END_VAR
IF iCam = 0 THEN
  Enable := FALSE;
  LogError('setCam failed: invalid reference');
ELSIF eState <> cL_IDLE THEN
  Enable := FALSE;
  LogError('enable failed: trigger busy');
ELSE
  iActiveCam := iCam;
  Enable     := TRUE;

  // save constant settings
  _bUseCameraTrigger := bUseCameraTrigger;
  _bUseCameraTriggerFeedback := bUseCameraTriggerFeedback;
END_IF;
END_METHOD

METHOD Init
VAR_INPUT
  nResolution                   : INT := 1;        (*Printhead Resolution [e.g. 600] x Subpixel Resolution [e.g. 32]*)
  bUsePositionTrigger           : BOOL;            (*FALSE: Calculate time with speed and position distance@sensor event*)
END_VAR
(*zero divisions*)
IF nResolution = 0 THEN 
  bInitOk :=FALSE;
  RETURN; 
END_IF;

_nResolution:=nResolution;
_bUsePositionTrigger :=bUsePositionTrigger;


bInitOk :=TRUE;
END_METHOD

(*
  Log timestamp difference (if verbose active).
  t1-t2 
*)
METHOD LogTsDiff : BOOL
VAR_INPUT
  aIdent : STRING;
  t1 : T_DCTIME64;
  t2 : T_DCTIME64;
END_VAR
IF _bVerbose THEN
  LogLvl(Lvl:=E_LogSeverity.Debug, Msg:=
       F_Concat7(aIdent, 
                 't1: ', TO_STRING(t1), 
                 ' t2: ', TO_STRING(t2), 
                 ' t1-t2 [ms]: ', TO_STRING((TO_LREAL(t1)-TO_LREAL(t2))*1E-6)
       )
  );
END_IF
END_METHOD

(*
  Detected start position X0 (absolute) in [SubPx].
*)
PROPERTY nStartPositionX0 : DINT
GET
nStartPositionX0 := _nX0;
END_GET
END_PROPERTY

METHOD Reset
VAR_INPUT
END_VAR
eState              := cL_IDLE;      // reset state
OtTriggerStartTime  := F_GetCurDcTaskTime64();  // now
ObTrigger           := FALSE;        // set output = 0
OnTriggerCommand    := nC_EL2252Cmd_ACTIVE;    // activate command
bInhibitTrigger := FALSE;
END_METHOD

METHOD SetSubstrateLength
VAR_INPUT
  fSubstrateLength : LREAL;
END_VAR
IF NOT bInitOk THEN RETURN;END_IF;

(*Added 10 mm margin for substrate length in case of print quality strips at the end of sheet in case of start with edge*)
_fSubstrateLength := fSubstrateLength + fC_SheetLengthMargin;
_nSubstrateLength := F_MeterToSubPixel(fPosMeter:=_fSubstrateLength, fResoSubPx:=_nResolution);
END_METHOD

END_FUNCTION_BLOCK

// ---- POUs/Print/Camera/FB_LineCamera.TcPOU
(*
  QualiVision line camera system
  Provides callback function (rx_callback) for received TcpIp messages.   
*)
FUNCTION_BLOCK FB_LineCamera EXTENDS FB_CameraTcpIp IMPLEMENTS I_Sim

VAR_INPUT
  InTempActValueScanner   AT%I* : INT;    (*Actual value temperature camera [0.1 C]*)
  InTempActValuePrintUnit       : INT;    (*Actual value temperature pu [0.1 C]*)
  IfSpeed                       : LREAL;  (*Actual speed [m/s]*)
END_VAR

VAR
  _fCameraWidthNormal       : LREAL;       (*cW: Camera width [m]*)
  _nCameraWidth             : DINT;        (*Camera width [px]*)
  _fCameraMechOffsetTC      : LREAL;       (*Camera mechanical offset at calibration temp [mm]*)
  _fMechOffsetCameraToPU    : LREAL;       (*Camera mechanical offset to PrintUnit [mm]*)
  _fPrintUnitMechOffsetTC   : LREAL;       (*PrintUnit mechanical offset at calibration temp [mm]*)
  _nPrintUnitWidthNormal    : UDINT;       (*Print unit width [px] native*)
  _fPrintUnitWidthTC        : LREAL;       (*pWc: Print unit width [m]*)
  _fPrintUnitCalTemp        : LREAL;       (*calibration temperature for the PrintUnit*)

  fCameraWidthTC            : LREAL;       (*cWc: Camera width [m] at specific calibration temperature*)
  fCameraTemp               : LREAL;       (*Camera actual temp [°C]*)
  fCameraDeltaTempFactor    : LREAL;       (*Factor for distance calculation at delta temp*)
  fCameraRealResolution     : LREAL;       (*real resolution (with the actual temperature) from the line camera in y direction*)
  fCameraMechOffsetTAct     : LREAL;       (*Camera mechanical offset at actual temp [mm]*)
  fCameraCenterOffsetTAct   : LREAL;       (*Camera center offset at actual temp [mm]*)
  
  fPrintUnitTemp            : LREAL;       (*PrintUnit actual temp [°C]*)
  fPrintUnitDeltaTempFactor : LREAL;       (*Factor for distance calculation at delta temp*)
  fPrintUnitMechOffsetTAct  : LREAL;       (*PrintUnit mechanical offset at actual temp [mm]*)
  fPrintUnitWidthTAct       : LREAL;       (*PrintUnit width at actual temp [mm]*)
  fPrintUnitWidthDiff       : LREAL;       (*PrintUnit width difference at actual temp [mm]*)
  fPrintUnitCenterOffsetTAct: LREAL;       (*PrintUnit center offset at actual temp [mm]*)

  fCameraDelay              : LREAL;      (*camera start delay from frame grabber (300dpi vs 600dpi phase sync.) in [m]*)            
  
  nNbVersion                : INT;
  sModus                    : T_MaxString;
  nSector                   : DINT;
  nNbMarks                  : UDINT;
  _bTeachOk                 : BOOL;
  nNbMarksTeach             : UDINT;
  nNbMarksScanned           : UDINT;
  nNbSectorTeach            : DINT;
  sTeach                    : T_MaxString;      // last teach message (255 chars only), for VISU only
  sCameraPoints             : ARRAY [1..GVL_Camera.cMaxNbMarks] OF ST_CameraPoint;   // camera points list of received 'A' frames, also used for 'T' at job start
  sTeachPoints              : ARRAY [1..GVL_Camera.cMaxNbMarks] OF ST_TeachPoint;    // teached points
  nNumPointsPerSectorT      : ARRAY [1..GVL_Camera.cMaxNbSectors] OF DINT;           // number of marks in theach in frame x
  nNumPointsPerSectorA      : ARRAY [1..GVL_Camera.cMaxNbSectors] OF DINT;           // number of marks received in frame x
  nNumFrames                : UDINT;                                      // number of camera frames for job
  
  // Messages
  fbMsg_NotEnoughTeachPoints  : FB_MESSAGE;
  bNotEnoughTeachPoints : BOOL;
  bNotAllFramesContainTeachPoints : BOOL;
  bInvalidTeachPointsReceived : BOOL;
  
  // debug ------------------------
  _bVerbose                 : BOOL;   // Enable verbose mode (log more debug information
  // camera timing
  // - loop test (PLC->QR->PLC)
  _bTestTx                  : BOOL; // send a message (loop time test) from VISU button
  _tTimeTx, _tTimeRx        : T_DCTIME64;
  _sTimeElapsed             : STRING;
  _tTimeTrigger             : T_DCTIME64;
  _nTimeFrameIdx_CamMsg     : UDINT := 1;
  _tTimeFrames_CamMsg       : ARRAY[0..nC_MaxRxTimingEntries] OF T_DCTIME64;   // TimeStamp of cam messages
  _tTimeFramesMs_CamMsg     : ARRAY[0..nC_MaxRxTimingEntries] OF LREAL;        // elapsed times of each frame since trigger
  _tTimeFrames_TestMsg      : ARRAY[0..nC_MaxRxTimingEntries] OF T_DCTIME64;   // TimeStamp of test messages
  _tTimeFramesMs_TestMsg    : ARRAY[0..nC_MaxRxTimingEntries] OF LREAL;        // elapsed time of each frame since trigger 
  // tcp camera simulation
  _nSimMode                 : UDINT := 0; // 0=generate points in plc, 1=use ext. cam simulation script, 2=send rx_callback messages directly
  _sSimCamPoints            : ARRAY [1..GVL_Camera.cMaxNbMarks] OF ST_DeformationPointAccurate;
  _nSimCamFrameDepth        : UDINT := 2048;   // distance of cam frames (point pitch in x in [px])
  _nSimCamMarksPerFrame     : UDINT := 6;  
  _bSimCamPointValid        : BOOL := TRUE;
  _aCamSimScriptPath        : T_MaxString;
  fbScriptCamSim            : FB_ScriptLauncher;    // external cam simulation script
  _rfTrigSim                : RF_TRIG;
//  _tStartSim                : TON;
  // ---- NOTE: vars accesses by CameraSimulation script, edit on both sides
  nScriptPID                : UDINT;
  nFrameNr                  : UDINT;
  // -----
END_VAR                     

VAR CONSTANT
  // protocol
  cErrorString              : T_MaxString := '<Error(';  (*not used yet*)
  cStartString              : T_MaxString := '<position(';
  cEndingString             : T_MaxString := ');';
  cProtoVersion_100         : INT := 100;               // initial protocol version
  cProtoVersion_110         : INT := 110;               // protocol extension +sector indication in T and A +end sector indication
  cIdxFirstSector           : UDINT := 1;
  
  // camera
  cCameraMinXY              : DINT := 0;       (*[px/4800dpi]*)
  cCameraMaxXY              : DINT := 205_000; (*[px/4800dpi]*)
  cCameraResolution         : LREAL := 300;     (*Camera pixel resolution [dpi]*)
  cCameraResolutionSubpixel : LREAL :=  16;     (*Subpixel point resolution [SubPx] -> 4800dpi*)
  cCameraTempCoefficient    : LREAL := 23.1E-6; (*thermal expansion coefficient from aluminium [1/K]*)
  // print unit
  cPrintUnitTempCoefficient : LREAL := 17.3E-6; (*thermal expansion coefficient from print unit base plate [1/K]*)
  fC_PhPixelDistFactorAtRefTemp: LREAL := 0.1693/4;(*RICOH GEN5 PH pixel distance [mm] y direction of one pixel at reference temperature (instead of native resolution 600dpi)*)
  fC_PhPixelDistRefTemp     : LREAL := 23;      (*RICOH GEN5 PH reference temperature matching the fC_PhPixelDistFactorAtRefTemp*)

  // test telegram definitions
  sQvTest_Header            : STRING := 'QT_'; // qualivision test telegram header
  sQvTest_CI                : STRING := 'CI_'; // input frame timing test
  sQvTest_Loop              : STRING := 'LP_'; // loop timing test
  
  // debug
  nC_MaxRxTimingEntries     : UDINT := 40;
END_VAR

VAR PERSISTENT
  fCameraResolution         : LREAL := cCameraResolution;  (*Camera pixel resolution [dpi]*)
  fCameraAdjustmentY        : LREAL := 0;            (*Camera adjustment in Y direction [mm]*)
  fCameraCalTemp            : LREAL := 25;           (*calibration temperature for the given line camera resolution*)    
  fCameraStartMargin        : LREAL := 0.0085;       (*cM: Camera start margin [m]*)
END_VAR

// - live configuration update & checks
// -- trigger, cam position and trigger settings (Worker position setup)
_fTriggerDistance    := _fDetectToCameraOffset - fCameraStartMargin;
IF IfSpeed <> 0 THEN
  _fTriggerPulseLength := (fSubstrateLength + 2*fCameraStartMargin) / IfSpeed * 1000;  (*[ms] Margin at start and end of the sheet*)
END_IF

// --
IF fCameraResolution > 0 THEN
  fCameraWidthTC := DINT_TO_LREAL(_nCameraWidth) / fCameraResolution * 0.0254;
ELSE
  fCameraWidthTC := FC_CONV_SUBPX_TO_M( _nCameraWidth, LREAL_TO_UDINT(cCameraResolution), 1);
END_IF;

(*Camera temperature compensation (y-pos, center and resolution)*)
fCameraTemp             := INT_TO_LREAL(InTempActValueScanner) * 0.1;
fCameraDeltaTempFactor  := 1 + (cCameraTempCoefficient * (fCameraTemp - fCameraCalTemp));
fCameraRealResolution   := fCameraResolution / fCameraDeltaTempFactor; 
fCameraMechOffsetTAct   := _fCameraMechOffsetTC * fCameraDeltaTempFactor;
fCameraCenterOffsetTAct := (((fCameraWidthTC / 2 * 1000) + _fCameraMechOffsetTC) * fCameraDeltaTempFactor) - ((fCameraWidthTC / 2 * 1000) + _fCameraMechOffsetTC);

fPrintUnitTemp             := INT_TO_LREAL(InTempActValuePrintUnit) * 0.1;
fPrintUnitDeltaTempFactor  := 1 + (cPrintUnitTempCoefficient * (fPrintUnitTemp - _fPrintUnitCalTemp));
fPrintUnitMechOffsetTAct   := _fPrintUnitMechOffsetTC * fPrintUnitDeltaTempFactor;
fPrintUnitWidthTAct        := _fPrintUnitWidthTC * fPrintUnitDeltaTempFactor;

fPrintUnitWidthDiff        := fPrintUnitWidthTAct - _fPrintUnitWidthTC;
fPrintUnitCenterOffsetTAct := (((_fPrintUnitWidthTC / 2 * 1000) + _fPrintUnitMechOffsetTC) * fPrintUnitDeltaTempFactor) - ((_fPrintUnitWidthTC / 2 * 1000) + _fPrintUnitMechOffsetTC);

SimUpdate();

// Messages
(*fbMsg_NotEnoughTeachPoints( bI_Status:=SEL(_bActivated, FALSE, bNotEnoughTeachPoints), 
                             iI_MsgNumber:=eC_DMAX_CAM_NOTENGOUGH_TEACH_POINTS, 
                             iI_MsgLocation:=ePr_BLK_CAMERA,
                             pI_MsgConfig:=_pMsgConfig);
*)

METHOD PRIVATE binarySearch : DINT
VAR_INPUT
  nLow : DINT;     // range lower
  nHigh : DINT;    // range upper
  nKey  : DINT;    // key to search
END_VAR
VAR
  mid : DINT;
END_VAR
IF nHigh < nLow THEN
  binarySearch := -1;
  RETURN;
END_IF

// split array in half
mid := (nLow + nHigh) / 2; (*low + (high - low)/2;*)

// did we find it?
IF nKey = TO_DINT(sTeachPoints[mid].id) THEN
  binarySearch := mid;
  RETURN;
END_IF

// no, search upper half (recursive)
IF nKey > TO_DINT(sTeachPoints[mid].id) THEN
  binarySearch := THIS^.binarySearch((mid + 1), nHigh, nKey);
  RETURN;
END_IF

// no, search lower half (recursive)
binarySearch:= THIS^.binarySearch(nLow, (mid - 1), nKey);
END_METHOD

{attribute 'monitoring' := 'call'}
(*Simulation is enabled set/get*)
PROPERTY bSimEnable : BOOL
GET
bSimEnable:=_bSimulate;
END_GET
SET
_bSimulate:=bSimEnable;
END_SET
END_PROPERTY

(*
  Calculate teached/saved reference points in print system coordinates.
*)
METHOD PRIVATE calcTeachPoints
VAR
  nCounter  : UDINT;
  nCurrSect : DINT;
  x_ref_abs : LREAL;
  y_ref_abs : LREAL;
  sTP       : ST_TeachPoint;
  sTPSend   : ST_DeformationPointAccurate;
END_VAR
IF _bVerbose THEN LogLvl(Lvl:=E_LogSeverity.Debug, Msg:='calculateTeachPoints()'); END_IF

bInvalidTeachPointsReceived := FALSE;

(*-- sort list with camera/teach points for faster binary searching later*)
sortPoints();

(*-- convert & save teach point in table separate table for later use*)
FOR nCounter := 1 TO nNbMarksTeach DO
  //--- save id
  sTP.id := sCameraPoints[nCounter].id;
  sTP.valid := sCameraPoints[nCounter].valid;
  
  //--- translate to print system coordinate system 
  IF (sCameraPoints[nCounter].x_ref = 0) THEN
    (*Fully automatic mode: ref value from camera is zero, ref value for printer is set with x.*)
    sTP.y_ref_Print   :=   ((_fPrintUnitWidthTC/2 + _fCameraWidthNormal/2) * 1000)  (*[m] => [mm]*)
                         - (  DINT_TO_REAL(sCameraPoints[nCounter].x)
                            / (cCameraResolution * cCameraResolutionSubpixel) * 25.4)           (*[mm]*)
                         - ((_fCameraWidthNormal - LREAL_TO_REAL(_fImageWidth)) * 1000 / 2);     (*[m] => [mm]*)
    sTP.y_teach_Print := 0;
  ELSE
    (*Semi automatic mode: ref value for printer is calculated with ref value and lx from camera.*)
    sTP.y_ref_Print   :=   (DINT_TO_REAL(sCameraPoints[nCounter].x_ref  - sCameraPoints[nCounter].lx)
                                      / (fCameraRealResolution * cCameraResolutionSubpixel) * 25.4);  (*[mm]*)
    sTP.y_teach_Print :=   (DINT_TO_REAL(sCameraPoints[nCounter].x)
                                      / (fCameraRealResolution * cCameraResolutionSubpixel) * 25.4);  (*[mm]*)
  END_IF
  
  IF (sCameraPoints[nCounter].y_ref = 0) THEN
    (*Fully automatic mode: ref value from camera is zero, ref value for printer is set with y.*)
    sTP.x_ref_Print   :=   (FC_CONV_SUBPX_TO_M( sCameraPoints[nCounter].y
                                              , LREAL_TO_UDINT(cCameraResolution)
                                              , LREAL_TO_UDINT(cCameraResolutionSubpixel)) * 1000)  (*[m] => [mm]*)
                         + (fCameraStartMargin * 1000);  (*[m] => [mm]*)
    sTP.x_teach_Print := 0;
  ELSE
    (*Semi automatic mode: ref value for printer is calculated with ref value and ly from camera.*)
    sTP.x_ref_Print   :=   (FC_CONV_SUBPX_TO_M( (sCameraPoints[nCounter].y_ref - sCameraPoints[nCounter].ly)
                                              , LREAL_TO_UDINT(cCameraResolution)
                                              , LREAL_TO_UDINT(cCameraResolutionSubpixel)) * 1000);  (*[m] => [mm]*)
    sTP.x_teach_Print :=   (FC_CONV_SUBPX_TO_M( sCameraPoints[nCounter].y
                                              , LREAL_TO_UDINT(cCameraResolution)
                                              , LREAL_TO_UDINT(cCameraResolutionSubpixel)) * 1000);  (*[m] => [mm]*)
  END_IF;
  
  //--- save teach point locally to seperate teach point array (the other one will be used for cam points while receiving) 
  sTeachPoints[nCounter] := sTP;
  
  //--- count points per sector (for error handling)
  IF (sTP.x_teach_Print = 0) THEN    (*Fully Automatic*)
    x_ref_abs := sTP.x_ref_Print;
  ELSE                                           (*Semi-automatic*)        
    x_ref_abs := sTP.x_ref_Print + sTP.x_teach_Print; 
  END_IF
  IF (sTP.y_teach_Print = 0) THEN    (*Fully Automatic*)
    y_ref_abs := sTP.y_ref_Print;
  ELSE                                           (*Semi-automatic*)        
    y_ref_abs := sTP.y_ref_Print + sTP.y_teach_Print;
  END_IF
  
  IF _fFrameLength <> 0 THEN
    nCurrSect := FC_LREAL_TO_DINT(x_ref_abs / _fFrameLength) + 1;
    nNumPointsPerSectorT[nCurrSect] := nNumPointsPerSectorT[nCurrSect] + 1;
  END_IF
  
  //--- send teach point to sink (python script)
  IF _iCameraSink <> 0 THEN
    sTPSend.x_ref := x_ref_abs;
    sTPSend.y_ref := y_ref_abs;
    sTPSend.dx    := 0;
    sTPSend.dy    := 0;
    sTPSend.col := nNumPointsPerSectorT[nCurrSect];  // point number in frame
    sTPSend.row := nCurrSect;                        // frame number
    _iCameraSink.AddTeachPoint(sTeachPoint:=sTPSend);
  END_IF
  
  //--- check if every teach point is valid
  IF NOT sTP.valid THEN
    bInvalidTeachPointsReceived := TRUE;
	END_IF
  
END_FOR

// verify the teach
verifyTeachPoints();
END_METHOD

METHOD CamTrigger
VAR_INPUT
  bOk             : BOOL;     // trigger is ok
	nPos            : DINT;     // camera triggered position
  nPosDeviation   : DINT;     // camera started deviation
  nX0             : DINT;     // detected position sheet/repetition
END_VAR
SUPER^.CamTrigger(bOk:=bOk, nPos:=nPos, nPosDeviation:=nPosDeviation, nX0:=nX0);

_tTimeTrigger := F_GetCurDcTaskTime64();    // save trigger time stamp (a little later than the real)
IF _bVerbose THEN LogLvl(Lvl:=E_LogSeverity.Debug, Msg:=F_Concat2('CamTrigger at: ', TO_STRING(_tTimeTrigger))); END_IF
nNbMarksScanned := 0;
END_METHOD

METHOD CamTriggerDone
SUPER^.CamTriggerDone();
IF _bVerbose THEN LogLvl(Lvl:=E_LogSeverity.Debug, Msg:=F_Concat2('CamTriggerDone at: ', TO_STRING(_tTimeTrigger))); END_IF
SimExit();
END_METHOD

(*
  Simulate camera points.
*)
METHOD PRIVATE CreateSimCamPoints : BOOL
VAR
  fbTonTimer     : TON;
  nCounter       : UDINT;
  nCamGridHeight : UDINT;    // cam points pitch in y in [px]
  nCamGridDepth  : UDINT;
  nIndex         : UDINT;
  nOffsetY       : UDINT;
  nCtr           : UDINT;
END_VAR
nCamGridDepth := _nSimCamFrameDepth;
nNbMarksTeach := _nSimCamMarksPerFrame * TO_UDINT((SEL(fSubstrateLength<>0, 5*nCamGridDepth, DINT_TO_UDINT(F_MeterToSubPixel(fPosMeter:=fSubstrateLength, fResoSubPx:=_nPrintUnitResolution)))) / nCamGridDepth);
nCamGridHeight := SEL(fSubstrateWidth<>0, 200, DINT_TO_UDINT(F_MeterToSubPixel(fPosMeter:=fSubstrateWidth, fResoSubPx:=_nPrintUnitResolution))/_nSimCamMarksPerFrame);
_bTeachOk := TRUE;

(*Test points*)
nCtr := 0;
nNbMarks := nNbMarksTeach;
nOffsetY := (_nPrintUnitWidthNormal-TO_UDINT(F_MeterToSubPixel(fPosMeter:=_fImageWidth, fResoSubPx:=_nPrintUnitResolution)))/2;

FOR nCounter := 0 TO nNbMarksTeach/_nSimCamMarksPerFrame - 1 DO    // col
  FOR nIndex := 0 TO _nSimCamMarksPerFrame-1 DO  // row
    // create point
    stCamPoint := getSimCamPoint(
      fOffsetMin:=-5.0,
      fOffsetMax:=5.0,
      fXMin:=nCounter*nCamGridDepth,
      fXMax:=(nCounter+1)*nCamGridDepth,
      fYMin:=nIndex*nCamGridHeight+nOffsetY,
      fYMax:=(nIndex+1)*nCamGridHeight+nOffsetY
    );
    // save simulation cam point
    nCtr := nCtr + 1;
    stCamPoint.index := TO_DINT(nCtr);
    stCamPoint.col   := TO_DINT(nCounter);
    stCamPoint.row   := TO_DINT(nIndex);
    _sSimCamPoints[nCtr] := stCamPoint;
  END_FOR
END_FOR
END_METHOD

{attribute 'monitoring':='call'}
PROPERTY eCameraMode : E_CameraMode
GET
// return active mode (after teach or live
eCameraMode := _eCameraMode;  // mode set by PUC

IF    _eCameraMode = E_CameraMode.Auto THEN
  eCameraMode := _ePossibleMode;
ELSIF _ePossibleMode < _eCameraMode THEN
  // reduced level
  eCameraMode := _ePossibleMode;
END_IF
END_GET
END_PROPERTY

PROPERTY eDeviceType : E_CameraDevice
GET
eDeviceType := E_CameraDevice.Scanner;
END_GET
END_PROPERTY

